      $ 3392 "'desbaste_inicial'"
      # 'desbaste_inicial'
      $ 3393 "bajada_broca≔p[0,0,-0.008,0,0,0]"
      global bajada_broca=p[0,0,-0.008,0,0,0]
      $ 3394 "bajada≔p[0,0,0.008,0,0,0]"
      global bajada=p[0,0,0.008,0,0,0]
      $ 3395 "Direction: Base Z-"
      global move_thread_flag_3395=0
      thread move_thread_3395():
        enter_critical
        move_thread_flag_3395 = 1
        local towardsPos=calculate_point_to_move_towards(p[0.0,0.0,0.0,0.0,0.0,0.0], [0.0,0.0,-1.0], 0.08)
        movel(towardsPos, a=0.035, v=0.03)
        move_thread_flag_3395 = 2
        exit_critical
      end
      move_thread_flag_3395 = 0
      move_thread_han_3395 = run move_thread_3395()
      while (True):
        sleep(1.0E-10)
        if (move_thread_flag_3395 > 1):
          join move_thread_han_3395
          $ 3396 "Until (distance)"
          break
        end
        sync()
      end
      $ 3397 "Popup: punto contacto alanzdo"
      popup("punto contacto alanzdo", "Mensaje", False, False, blocking=True)
      $ 3398 "Direction: Base Z+"
      global move_thread_flag_3398=0
      thread move_thread_3398():
        enter_critical
        move_thread_flag_3398 = 1
        local towardsPos=calculate_point_to_move_towards(p[0.0,0.0,0.0,0.0,0.0,0.0], [0.0,0.0,1.0], 0.002)
        movel(towardsPos, a=0.005, v=0.003)
        move_thread_flag_3398 = 2
        exit_critical
      end
      move_thread_flag_3398 = 0
      move_thread_han_3398 = run move_thread_3398()
      while (True):
        sleep(1.0E-10)
        if (move_thread_flag_3398 > 1):
          join move_thread_han_3398
          $ 3399 "Until (distance)"
          break
        end
        sync()
      end
      $ 3400 "Wait: 0.3"
      sleep(0.3)
      $ 3401 "Set CO[1]=Encender"
      set_configurable_digital_out(1, True)
      $ 3402 "Wait: 0.3"
      sleep(0.3)
      $ 3403 "Loop 3 times"
      Loop_58 = 0
      while (Loop_58 < 3):
        $ 3404 "bajar≔pose_add(get_actual_tcp_pose(), bajada_broca)"
        global bajar= pose_add ( get_actual_tcp_pose (), bajada_broca)
        $ 3405 "bajar" "breakAfter"
        movel(bajar, a=0.005, v=0.001)
        $ 3406 "subir≔pose_sub(get_actual_tcp_pose(), bajada_broca)"
        global subir= pose_sub ( get_actual_tcp_pose (), bajada_broca)
        $ 3407 "subir" "breakAfter"
        movel(subir, a=0.01, v=0.01)
        $ 3408 "bajada_broca≔pose_sub(bajada_broca, bajada)"
        global bajada_broca= pose_sub (bajada_broca, bajada)
        Loop_58 = Loop_58 + 1
      end
      $ 3409 "Direction: Base Z+"
      global move_thread_flag_3409=0
      thread move_thread_3409():
        enter_critical
        move_thread_flag_3409 = 1
        local towardsPos=calculate_point_to_move_towards(p[0.0,0.0,0.0,0.0,0.0,0.0], [0.0,0.0,1.0], 0.06)
        movel(towardsPos, a=0.035, v=0.03)
        move_thread_flag_3409 = 2
        exit_critical
      end
      move_thread_flag_3409 = 0
      move_thread_han_3409 = run move_thread_3409()
      while (True):
        sleep(1.0E-10)
        if (move_thread_flag_3409 > 1):
          join move_thread_han_3409
          $ 3410 "Until (distance)"
          break
        end
        sync()
      end
      $ 3411 "Set CO[1]=Apagar"
      set_configurable_digital_out(1, False)
      $ 3412 "barreno_actual≔barreno_actual+1"
      global barreno_actual=barreno_actual+1
      $ 3413 "If barreno_actual>barrenos_menos1"
      if (barreno_actual>barrenos_menos1):
        $ 3414 "cambiar_broca≔ True "
        global cambiar_broca=  True
      end
      $ 3415 "Call Quitar_broca"
      Quitar_broca()
      $ 3416 "Call Poner_broca"
      Poner_broca()
    end
    $ 3417 "Popup: Linea4 con chica Terminada!"
    popup("Linea4 con chica Terminada!", "Mensaje", False, False, blocking=True)
    $ 3418 "Broca_2"
    $ 3419 "Linea3"
    $ 3420 "Marcar_puntos"
    $ 3421 "MoveL"
    $ 3422 "Home3" "breakAfter"
    movel(Home3_p, a=0.5, v=0.1)
    $ 3423 "Linea3_A" "breakAfter"
    movel(Linea3_A_p, a=0.5, v=0.1)
    $ 3424 "Linea3_B" "breakAfter"
    movel(Linea3_B_p, a=0.5, v=0.1)
    $ 3425 "Linea3_C" "breakAfter"
    movel(Linea3_C_p, a=0.5, v=0.1)
    $ 3426 "Linea3_D" "breakAfter"
    movel(Linea3_D_p, a=0.5, v=0.1)
    $ 3427 "Linea3_E" "breakAfter"
    movel(Linea3_E_p, a=0.5, v=0.1)
    $ 3428 "Linea3_F" "breakAfter"
    movel(Linea3_F_p, a=0.5, v=0.1)
    $ 3429 "AB"
    $ 3430 "'desbaste_inicial'"
    # 'desbaste_inicial'
    $ 3431 "bajada_broca≔p[0,0,-0.012,0,0,0]"
    global bajada_broca=p[0,0,-0.012,0,0,0]
    $ 3432 "barrenos_menos1≔8"
    global barrenos_menos1=8
    $ 3433 "barreno_actual≔0"
    global barreno_actual=0
    $ 3434 "Loop barreno_actual≤barrenos_menos1"
    while (barreno_actual <= barrenos_menos1):
      $ 3435 "Perforacion"
      $ 3436 "MoveL"
      $ 3437 "internos≔interpolate_pose(Linea3_A, Linea3_B, barreno_actual/barrenos_menos1)"
      global internos= interpolate_pose (Linea3_A_p, Linea3_B_p, barreno_actual/barrenos_menos1)
      $ 3438 "internos" "breakAfter"
      movel(internos, a=0.5, v=0.1)
      $ 3439 "'desbaste_inicial'"
      # 'desbaste_inicial'
      $ 3440 "bajada_broca≔p[0,0,-0.012,0,0,0]"
      global bajada_broca=p[0,0,-0.012,0,0,0]
      $ 3441 "bajada≔p[0,0,0.012,0,0,0]"
      global bajada=p[0,0,0.012,0,0,0]
      $ 3442 "Direction: Base Z-"
      global move_thread_flag_3442=0
      thread move_thread_3442():
        enter_critical
        move_thread_flag_3442 = 1
        local towardsPos=calculate_point_to_move_towards(p[0.0,0.0,0.0,0.0,0.0,0.0], [0.0,0.0,-1.0], 0.08)
        movel(towardsPos, a=0.035, v=0.03)
        move_thread_flag_3442 = 2
        exit_critical
      end
      move_thread_flag_3442 = 0
      move_thread_han_3442 = run move_thread_3442()
      while (True):
        sleep(1.0E-10)
        if (move_thread_flag_3442 > 1):
          join move_thread_han_3442
          $ 3443 "Until (distance)"
          break
        end
        sync()
      end
      $ 3444 "Popup: punto contacto alanzdo"
      popup("punto contacto alanzdo", "Mensaje", False, False, blocking=True)
      $ 3445 "Direction: Base Z+"
      global move_thread_flag_3445=0
      thread move_thread_3445():
        enter_critical
        move_thread_flag_3445 = 1
        local towardsPos=calculate_point_to_move_towards(p[0.0,0.0,0.0,0.0,0.0,0.0], [0.0,0.0,1.0], 0.002)
        movel(towardsPos, a=0.005, v=0.003)
        move_thread_flag_3445 = 2
        exit_critical
      end
      move_thread_flag_3445 = 0
      move_thread_han_3445 = run move_thread_3445()
      while (True):
        sleep(1.0E-10)
        if (move_thread_flag_3445 > 1):
          join move_thread_han_3445
          $ 3446 "Until (distance)"
          break
        end
        sync()
      end
      $ 3447 "Wait: 0.3"
      sleep(0.3)
      $ 3448 "Set CO[1]=Encender"
      set_configurable_digital_out(1, True)
      $ 3449 "Wait: 0.3"
      sleep(0.3)
      $ 3450 "Loop 2 times"
      Loop_60 = 0
      while (Loop_60 < 2):
        $ 3451 "bajar≔pose_add(get_actual_tcp_pose(), bajada_broca)"
        global bajar= pose_add ( get_actual_tcp_pose (), bajada_broca)
        $ 3452 "bajar" "breakAfter"
        movel(bajar, a=0.005, v=0.001)
        $ 3453 "subir≔pose_sub(get_actual_tcp_pose(), bajada_broca)"
        global subir= pose_sub ( get_actual_tcp_pose (), bajada_broca)
        $ 3454 "subir" "breakAfter"
        movel(subir, a=0.01, v=0.01)
        $ 3455 "bajada_broca≔pose_sub(bajada_broca, bajada)"
        global bajada_broca= pose_sub (bajada_broca, bajada)
        Loop_60 = Loop_60 + 1
      end
      $ 3456 "Direction: Base Z+"
      global move_thread_flag_3456=0
      thread move_thread_3456():
        enter_critical
        move_thread_flag_3456 = 1
        local towardsPos=calculate_point_to_move_towards(p[0.0,0.0,0.0,0.0,0.0,0.0], [0.0,0.0,1.0], 0.06)
        movel(towardsPos, a=0.035, v=0.03)
        move_thread_flag_3456 = 2
        exit_critical
      end
      move_thread_flag_3456 = 0
      move_thread_han_3456 = run move_thread_3456()
      while (True):
        sleep(1.0E-10)
        if (move_thread_flag_3456 > 1):
          join move_thread_han_3456
          $ 3457 "Until (distance)"
          break
        end
        sync()
      end
      $ 3458 "Set CO[1]=Apagar"
      set_configurable_digital_out(1, False)
      $ 3459 "barreno_actual≔barreno_actual+1"
      global barreno_actual=barreno_actual+1
      $ 3460 "Call Quitar_broca"
      Quitar_broca()
      $ 3461 "Call Poner_broca"
      Poner_broca()
    end
    $ 3462 "CD"
    $ 3463 "'desbaste_inicial'"
    # 'desbaste_inicial'
    $ 3464 "bajada_broca≔p[0,0,-0.012,0,0,0]"
    global bajada_broca=p[0,0,-0.012,0,0,0]
    $ 3465 "barrenos_menos1≔8"
    global barrenos_menos1=8
    $ 3466 "barreno_actual≔0"
    global barreno_actual=0
    $ 3467 "Loop barreno_actual≤barrenos_menos1"
    while (barreno_actual <= barrenos_menos1):
      $ 3468 "Perforacion"
      $ 3469 "MoveL"
      $ 3470 "internos≔interpolate_pose(Linea3_C, Linea3_D, barreno_actual/barrenos_menos1)"
      global internos= interpolate_pose (Linea3_C_p, Linea3_D_p, barreno_actual/barrenos_menos1)
      $ 3471 "internos" "breakAfter"
      movel(internos, a=0.5, v=0.1)
      $ 3472 "'desbaste_inicial'"
      # 'desbaste_inicial'
      $ 3473 "bajada_broca≔p[0,0,-0.012,0,0,0]"
      global bajada_broca=p[0,0,-0.012,0,0,0]
      $ 3474 "bajada≔p[0,0,0.012,0,0,0]"
      global bajada=p[0,0,0.012,0,0,0]
      $ 3475 "Direction: Base Z-"
      global move_thread_flag_3475=0
      thread move_thread_3475():
        enter_critical
        move_thread_flag_3475 = 1
        local towardsPos=calculate_point_to_move_towards(p[0.0,0.0,0.0,0.0,0.0,0.0], [0.0,0.0,-1.0], 0.08)
        movel(towardsPos, a=0.035, v=0.03)
        move_thread_flag_3475 = 2
        exit_critical
      end
      move_thread_flag_3475 = 0
      move_thread_han_3475 = run move_thread_3475()
      while (True):
        sleep(1.0E-10)
        if (move_thread_flag_3475 > 1):
          join move_thread_han_3475
          $ 3476 "Until (distance)"
          break
        end
        sync()
      end
      $ 3477 "Popup: punto contacto alanzdo"
      popup("punto contacto alanzdo", "Mensaje", False, False, blocking=True)
      $ 3478 "Direction: Base Z+"
      global move_thread_flag_3478=0
      thread move_thread_3478():
        enter_critical
        move_thread_flag_3478 = 1
        local towardsPos=calculate_point_to_move_towards(p[0.0,0.0,0.0,0.0,0.0,0.0], [0.0,0.0,1.0], 0.002)
        movel(towardsPos, a=0.005, v=0.003)
        move_thread_flag_3478 = 2
        exit_critical
      end
      move_thread_flag_3478 = 0
      move_thread_han_3478 = run move_thread_3478()
      while (True):
        sleep(1.0E-10)
        if (move_thread_flag_3478 > 1):
          join move_thread_han_3478
          $ 3479 "Until (distance)"
          break
        end
        sync()
      end
      $ 3480 "Wait: 0.3"
      sleep(0.3)
      $ 3481 "Set CO[1]=Encender"
      set_configurable_digital_out(1, True)
      $ 3482 "Wait: 0.3"
      sleep(0.3)
      $ 3483 "Loop 2 times"
      Loop_64 = 0
      while (Loop_64 < 2):
        $ 3484 "bajar≔pose_add(get_actual_tcp_pose(), bajada_broca)"
        global bajar= pose_add ( get_actual_tcp_pose (), bajada_broca)
        $ 3485 "bajar" "breakAfter"
        movel(bajar, a=0.005, v=0.001)
        $ 3486 "subir≔pose_sub(get_actual_tcp_pose(), bajada_broca)"
        global subir= pose_sub ( get_actual_tcp_pose (), bajada_broca)
        $ 3487 "subir" "breakAfter"
        movel(subir, a=0.01, v=0.01)
        $ 3488 "bajada_broca≔pose_sub(bajada_broca, bajada)"
        global bajada_broca= pose_sub (bajada_broca, bajada)
        Loop_64 = Loop_64 + 1
      end
      $ 3489 "Direction: Base Z+"
      global move_thread_flag_3489=0
      thread move_thread_3489():
        enter_critical
        move_thread_flag_3489 = 1
        local towardsPos=calculate_point_to_move_towards(p[0.0,0.0,0.0,0.0,0.0,0.0], [0.0,0.0,1.0], 0.06)
        movel(towardsPos, a=0.035, v=0.03)
        move_thread_flag_3489 = 2
        exit_critical
      end
      move_thread_flag_3489 = 0
      move_thread_han_3489 = run move_thread_3489()
      while (True):
        sleep(1.0E-10)
        if (move_thread_flag_3489 > 1):
          join move_thread_han_3489
          $ 3490 "Until (distance)"
          break
        end
        sync()
      end
      $ 3491 "Set CO[1]=Apagar"
      set_configurable_digital_out(1, False)
      $ 3492 "barreno_actual≔barreno_actual+1"
      global barreno_actual=barreno_actual+1
      $ 3493 "Call Quitar_broca"
      Quitar_broca()
      $ 3494 "Call Poner_broca"
      Poner_broca()
    end
    $ 3495 "EF"
    $ 3496 "'desbaste_inicial'"
    # 'desbaste_inicial'
    $ 3497 "bajada_broca≔p[0,0,-0.012,0,0,0]"
    global bajada_broca=p[0,0,-0.012,0,0,0]
    $ 3498 "barrenos_menos1≔8"
    global barrenos_menos1=8
    $ 3499 "barreno_actual≔0"
    global barreno_actual=0
    $ 3500 "Loop barreno_actual≤barrenos_menos1"
    while (barreno_actual <= barrenos_menos1):
      $ 3501 "Perforacion"
      $ 3502 "MoveL"
      $ 3503 "internos≔interpolate_pose(Linea3_E, Linea3_F, barreno_actual/barrenos_menos1)"
      global internos= interpolate_pose (Linea3_E_p, Linea3_F_p, barreno_actual/barrenos_menos1)
      $ 3504 "internos" "breakAfter"
      movel(internos, a=0.5, v=0.1)
      $ 3505 "'desbaste_inicial'"
      # 'desbaste_inicial'
      $ 3506 "bajada_broca≔p[0,0,-0.012,0,0,0]"
      global bajada_broca=p[0,0,-0.012,0,0,0]
      $ 3507 "bajada≔p[0,0,0.012,0,0,0]"
      global bajada=p[0,0,0.012,0,0,0]
      $ 3508 "Direction: Base Z-"
      global move_thread_flag_3508=0
      thread move_thread_3508():
        enter_critical
        move_thread_flag_3508 = 1
        local towardsPos=calculate_point_to_move_towards(p[0.0,0.0,0.0,0.0,0.0,0.0], [0.0,0.0,-1.0], 0.08)
        movel(towardsPos, a=0.035, v=0.03)
        move_thread_flag_3508 = 2
        exit_critical
      end
      move_thread_flag_3508 = 0
      move_thread_han_3508 = run move_thread_3508()
      while (True):
        sleep(1.0E-10)
        if (move_thread_flag_3508 > 1):
          join move_thread_han_3508
          $ 3509 "Until (distance)"
          break
        end
        sync()
      end
      $ 3510 "Popup: punto contacto alanzdo"
      popup("punto contacto alanzdo", "Mensaje", False, False, blocking=True)
      $ 3511 "Direction: Base Z+"
      global move_thread_flag_3511=0
      thread move_thread_3511():
        enter_critical
        move_thread_flag_3511 = 1
        local towardsPos=calculate_point_to_move_towards(p[0.0,0.0,0.0,0.0,0.0,0.0], [0.0,0.0,1.0], 0.002)
        movel(towardsPos, a=0.005, v=0.003)
        move_thread_flag_3511 = 2
        exit_critical
      end
      move_thread_flag_3511 = 0
      move_thread_han_3511 = run move_thread_3511()
      while (True):
        sleep(1.0E-10)
        if (move_thread_flag_3511 > 1):
          join move_thread_han_3511
          $ 3512 "Until (distance)"
          break
        end
        sync()
      end
      $ 3513 "Wait: 0.3"
      sleep(0.3)
      $ 3514 "Set CO[1]=Encender"
      set_configurable_digital_out(1, True)
      $ 3515 "Wait: 0.3"
      sleep(0.3)
      $ 3516 "Loop 2 times"
      Loop_68 = 0
      while (Loop_68 < 2):
        $ 3517 "bajar≔pose_add(get_actual_tcp_pose(), bajada_broca)"
        global bajar= pose_add ( get_actual_tcp_pose (), bajada_broca)
        $ 3518 "bajar" "breakAfter"
        movel(bajar, a=0.005, v=0.001)
        $ 3519 "subir≔pose_sub(get_actual_tcp_pose(), bajada_broca)"
        global subir= pose_sub ( get_actual_tcp_pose (), bajada_broca)
        $ 3520 "subir" "breakAfter"
        movel(subir, a=0.01, v=0.01)
        $ 3521 "bajada_broca≔pose_sub(bajada_broca, bajada)"
        global bajada_broca= pose_sub (bajada_broca, bajada)
        Loop_68 = Loop_68 + 1
      end
      $ 3522 "Direction: Base Z+"
      global move_thread_flag_3522=0
      thread move_thread_3522():
        enter_critical
        move_thread_flag_3522 = 1
        local towardsPos=calculate_point_to_move_towards(p[0.0,0.0,0.0,0.0,0.0,0.0], [0.0,0.0,1.0], 0.06)
        movel(towardsPos, a=0.035, v=0.03)
        move_thread_flag_3522 = 2
        exit_critical
      end
      move_thread_flag_3522 = 0
      move_thread_han_3522 = run move_thread_3522()
      while (True):
        sleep(1.0E-10)
        if (move_thread_flag_3522 > 1):
          join move_thread_han_3522
          $ 3523 "Until (distance)"
          break
        end
        sync()
      end
      $ 3524 "Set CO[1]=Apagar"
      set_configurable_digital_out(1, False)
      $ 3525 "barreno_actual≔barreno_actual+1"
      global barreno_actual=barreno_actual+1
      $ 3526 "Call Quitar_broca"
      Quitar_broca()
      $ 3527 "Call Poner_broca"
      Poner_broca()
    end
    $ 3528 "Popup: Linea3 con media Terminada!"
    popup("Linea3 con media Terminada!", "Mensaje", False, False, blocking=True)
    $ 3529 "Linea4"
    $ 3530 "Marcar_puntos"
    $ 3531 "MoveL"
    $ 3532 "Home3" "breakAfter"
    movel(Home3_p, a=0.5, v=0.1)
    $ 3533 "Linea4_A" "breakAfter"
    movel(Linea4_A_p, a=0.5, v=0.1)
    $ 3534 "Linea4_B" "breakAfter"
    movel(Linea4_B_p, a=0.5, v=0.1)
    $ 3535 "Linea4_C" "breakAfter"
    movel(Linea4_C_p, a=0.5, v=0.1)
    $ 3536 "Linea4_D" "breakAfter"
    movel(Linea4_D_p, a=0.5, v=0.1)
    $ 3537 "Linea4_E" "breakAfter"
    movel(Linea4_E_p, a=0.5, v=0.1)
    $ 3538 "Linea4_F" "breakAfter"
    movel(Linea4_F_p, a=0.5, v=0.1)
    $ 3539 "AB"
    $ 3540 "'desbaste_inicial'"
    # 'desbaste_inicial'
    $ 3541 "bajada_broca≔p[0,0,-0.012,0,0,0]"
    global bajada_broca=p[0,0,-0.012,0,0,0]
    $ 3542 "barrenos_menos1≔8"
    global barrenos_menos1=8
    $ 3543 "barreno_actual≔0"
    global barreno_actual=0
    $ 3544 "Loop barreno_actual≤barrenos_menos1"
    while (barreno_actual <= barrenos_menos1):
      $ 3545 "Perforacion"
      $ 3546 "MoveL"
      $ 3547 "internos≔interpolate_pose(Linea4_A, Linea4_B, barreno_actual/barrenos_menos1)"
      global internos= interpolate_pose (Linea4_A_p, Linea4_B_p, barreno_actual/barrenos_menos1)
      $ 3548 "internos" "breakAfter"
      movel(internos, a=0.5, v=0.1)
      $ 3549 "'desbaste_inicial'"
      # 'desbaste_inicial'
      $ 3550 "bajada_broca≔p[0,0,-0.012,0,0,0]"
      global bajada_broca=p[0,0,-0.012,0,0,0]
      $ 3551 "bajada≔p[0,0,0.012,0,0,0]"
      global bajada=p[0,0,0.012,0,0,0]
      $ 3552 "Direction: Base Z-"
      global move_thread_flag_3552=0
      thread move_thread_3552():
        enter_critical
        move_thread_flag_3552 = 1
        local towardsPos=calculate_point_to_move_towards(p[0.0,0.0,0.0,0.0,0.0,0.0], [0.0,0.0,-1.0], 0.08)
        movel(towardsPos, a=0.035, v=0.03)
        move_thread_flag_3552 = 2
        exit_critical
      end
      move_thread_flag_3552 = 0
      move_thread_han_3552 = run move_thread_3552()
      while (True):
        sleep(1.0E-10)
        if (move_thread_flag_3552 > 1):
          join move_thread_han_3552
          $ 3553 "Until (distance)"
          break
        end
        sync()
      end
      $ 3554 "Popup: punto contacto alanzdo"
      popup("punto contacto alanzdo", "Mensaje", False, False, blocking=True)
      $ 3555 "Direction: Base Z+"
      global move_thread_flag_3555=0
      thread move_thread_3555():
        enter_critical
        move_thread_flag_3555 = 1
        local towardsPos=calculate_point_to_move_towards(p[0.0,0.0,0.0,0.0,0.0,0.0], [0.0,0.0,1.0], 0.002)
        movel(towardsPos, a=0.005, v=0.003)
        move_thread_flag_3555 = 2
        exit_critical
      end
      move_thread_flag_3555 = 0
      move_thread_han_3555 = run move_thread_3555()
      while (True):
        sleep(1.0E-10)
        if (move_thread_flag_3555 > 1):
          join move_thread_han_3555
          $ 3556 "Until (distance)"
          break
        end
        sync()
      end
      $ 3557 "Wait: 0.3"
      sleep(0.3)
      $ 3558 "Set CO[1]=Encender"
      set_configurable_digital_out(1, True)
      $ 3559 "Wait: 0.3"
      sleep(0.3)
      $ 3560 "Loop 2 times"
      Loop_72 = 0
      while (Loop_72 < 2):
        $ 3561 "bajar≔pose_add(get_actual_tcp_pose(), bajada_broca)"
        global bajar= pose_add ( get_actual_tcp_pose (), bajada_broca)
        $ 3562 "bajar" "breakAfter"
        movel(bajar, a=0.005, v=0.001)
        $ 3563 "subir≔pose_sub(get_actual_tcp_pose(), bajada_broca)"
        global subir= pose_sub ( get_actual_tcp_pose (), bajada_broca)
        $ 3564 "subir" "breakAfter"
        movel(subir, a=0.01, v=0.01)
        $ 3565 "bajada_broca≔pose_sub(bajada_broca, bajada)"
        global bajada_broca= pose_sub (bajada_broca, bajada)
        Loop_72 = Loop_72 + 1
      end
      $ 3566 "Direction: Base Z+"
      global move_thread_flag_3566=0
      thread move_thread_3566():
        enter_critical
        move_thread_flag_3566 = 1
        local towardsPos=calculate_point_to_move_towards(p[0.0,0.0,0.0,0.0,0.0,0.0], [0.0,0.0,1.0], 0.06)
        movel(towardsPos, a=0.035, v=0.03)
        move_thread_flag_3566 = 2
        exit_critical
      end
      move_thread_flag_3566 = 0
      move_thread_han_3566 = run move_thread_3566()
      while (True):
        sleep(1.0E-10)
        if (move_thread_flag_3566 > 1):
          join move_thread_han_3566
          $ 3567 "Until (distance)"
          break
        end
        sync()
      end
      $ 3568 "Set CO[1]=Apagar"
      set_configurable_digital_out(1, False)
      $ 3569 "barreno_actual≔barreno_actual+1"
      global barreno_actual=barreno_actual+1
      $ 3570 "Call Quitar_broca"
      Quitar_broca()
      $ 3571 "Call Poner_broca"
      Poner_broca()
    end
    $ 3572 "CD"
    $ 3573 "'desbaste_inicial'"
    # 'desbaste_inicial'
    $ 3574 "bajada_broca≔p[0,0,-0.012,0,0,0]"
    global bajada_broca=p[0,0,-0.012,0,0,0]
    $ 3575 "barrenos_menos1≔8"
    global barrenos_menos1=8
    $ 3576 "barreno_actual≔0"
    global barreno_actual=0
    $ 3577 "Loop barreno_actual≤barrenos_menos1"
    while (barreno_actual <= barrenos_menos1):
      $ 3578 "Perforacion"
      $ 3579 "MoveL"
      $ 3580 "internos≔interpolate_pose(Linea4_C, Linea4_D, barreno_actual/barrenos_menos1)"
      global internos= interpolate_pose (Linea4_C_p, Linea4_D_p, barreno_actual/barrenos_menos1)
      $ 3581 "internos" "breakAfter"
      movel(internos, a=0.5, v=0.1)
      $ 3582 "'desbaste_inicial'"
      # 'desbaste_inicial'
      $ 3583 "bajada_broca≔p[0,0,-0.012,0,0,0]"
      global bajada_broca=p[0,0,-0.012,0,0,0]
      $ 3584 "bajada≔p[0,0,0.012,0,0,0]"
      global bajada=p[0,0,0.012,0,0,0]
      $ 3585 "Direction: Base Z-"
      global move_thread_flag_3585=0
      thread move_thread_3585():
        enter_critical
        move_thread_flag_3585 = 1
        local towardsPos=calculate_point_to_move_towards(p[0.0,0.0,0.0,0.0,0.0,0.0], [0.0,0.0,-1.0], 0.08)
        movel(towardsPos, a=0.035, v=0.03)
        move_thread_flag_3585 = 2
        exit_critical
      end
      move_thread_flag_3585 = 0
      move_thread_han_3585 = run move_thread_3585()
      while (True):
        sleep(1.0E-10)
        if (move_thread_flag_3585 > 1):
          join move_thread_han_3585
          $ 3586 "Until (distance)"
          break
        end
        sync()
      end
      $ 3587 "Popup: punto contacto alanzdo"
      popup("punto contacto alanzdo", "Mensaje", False, False, blocking=True)
      $ 3588 "Direction: Base Z+"
      global move_thread_flag_3588=0
      thread move_thread_3588():
        enter_critical
        move_thread_flag_3588 = 1
        local towardsPos=calculate_point_to_move_towards(p[0.0,0.0,0.0,0.0,0.0,0.0], [0.0,0.0,1.0], 0.002)
        movel(towardsPos, a=0.005, v=0.003)
        move_thread_flag_3588 = 2
        exit_critical
      end
      move_thread_flag_3588 = 0
      move_thread_han_3588 = run move_thread_3588()
      while (True):
        sleep(1.0E-10)
        if (move_thread_flag_3588 > 1):
          join move_thread_han_3588
          $ 3589 "Until (distance)"
          break
        end
        sync()
      end
      $ 3590 "Wait: 0.3"
      sleep(0.3)
      $ 3591 "Set CO[1]=Encender"
      set_configurable_digital_out(1, True)
      $ 3592 "Wait: 0.3"
      sleep(0.3)
      $ 3593 "Loop 2 times"
      Loop_77 = 0
      while (Loop_77 < 2):
        $ 3594 "bajar≔pose_add(get_actual_tcp_pose(), bajada_broca)"
        global bajar= pose_add ( get_actual_tcp_pose (), bajada_broca)
        $ 3595 "bajar" "breakAfter"
        movel(bajar, a=0.005, v=0.001)
        $ 3596 "subir≔pose_sub(get_actual_tcp_pose(), bajada_broca)"
        global subir= pose_sub ( get_actual_tcp_pose (), bajada_broca)
        $ 3597 "subir" "breakAfter"
        movel(subir, a=0.01, v=0.01)
        $ 3598 "bajada_broca≔pose_sub(bajada_broca, bajada)"
        global bajada_broca= pose_sub (bajada_broca, bajada)
        Loop_77 = Loop_77 + 1
      end
      $ 3599 "Direction: Base Z+"
      global move_thread_flag_3599=0
      thread move_thread_3599():
        enter_critical
        move_thread_flag_3599 = 1
        local towardsPos=calculate_point_to_move_towards(p[0.0,0.0,0.0,0.0,0.0,0.0], [0.0,0.0,1.0], 0.06)
        movel(towardsPos, a=0.035, v=0.03)
        move_thread_flag_3599 = 2
        exit_critical
      end
      move_thread_flag_3599 = 0
      move_thread_han_3599 = run move_thread_3599()
      while (True):
        sleep(1.0E-10)
        if (move_thread_flag_3599 > 1):
          join move_thread_han_3599
          $ 3600 "Until (distance)"
          break
        end
        sync()
      end
      $ 3601 "Set CO[1]=Apagar"
      set_configurable_digital_out(1, False)
      $ 3602 "barreno_actual≔barreno_actual+1"
      global barreno_actual=barreno_actual+1
      $ 3603 "Call Quitar_broca"
      Quitar_broca()
      $ 3604 "Call Poner_broca"
      Poner_broca()
    end
    $ 3605 "EF"
    $ 3606 "'desbaste_inicial'"
    # 'desbaste_inicial'
    $ 3607 "bajada_broca≔p[0,0,-0.012,0,0,0]"
    global bajada_broca=p[0,0,-0.012,0,0,0]
    $ 3608 "barrenos_menos1≔8"
    global barrenos_menos1=8
    $ 3609 "barreno_actual≔0"
    global barreno_actual=0
    $ 3610 "Loop barreno_actual≤barrenos_menos1"
    while (barreno_actual <= barrenos_menos1):
      $ 3611 "Perforacion"
      $ 3612 "MoveL"
      $ 3613 "internos≔interpolate_pose(Linea4_E, Linea4_F, barreno_actual/barrenos_menos1)"
      global internos= interpolate_pose (Linea4_E_p, Linea4_F_p, barreno_actual/barrenos_menos1)
      $ 3614 "internos" "breakAfter"
      movel(internos, a=0.5, v=0.1)
      $ 3615 "'desbaste_inicial'"
      # 'desbaste_inicial'
      $ 3616 "bajada_broca≔p[0,0,-0.012,0,0,0]"
      global bajada_broca=p[0,0,-0.012,0,0,0]
      $ 3617 "bajada≔p[0,0,0.012,0,0,0]"
      global bajada=p[0,0,0.012,0,0,0]
      $ 3618 "Direction: Base Z-"
      global move_thread_flag_3618=0
      thread move_thread_3618():
        enter_critical
        move_thread_flag_3618 = 1
        local towardsPos=calculate_point_to_move_towards(p[0.0,0.0,0.0,0.0,0.0,0.0], [0.0,0.0,-1.0], 0.08)
        movel(towardsPos, a=0.035, v=0.03)
        move_thread_flag_3618 = 2
        exit_critical
      end
      move_thread_flag_3618 = 0
      move_thread_han_3618 = run move_thread_3618()
      while (True):
        sleep(1.0E-10)
        if (move_thread_flag_3618 > 1):
          join move_thread_han_3618
          $ 3619 "Until (distance)"
          break
        end
        sync()
      end
      $ 3620 "Popup: punto contacto alanzdo"
      popup("punto contacto alanzdo", "Mensaje", False, False, blocking=True)
      $ 3621 "Direction: Base Z+"
      global move_thread_flag_3621=0
      thread move_thread_3621():
        enter_critical
        move_thread_flag_3621 = 1
        local towardsPos=calculate_point_to_move_towards(p[0.0,0.0,0.0,0.0,0.0,0.0], [0.0,0.0,1.0], 0.002)
        movel(towardsPos, a=0.005, v=0.003)
        move_thread_flag_3621 = 2
        exit_critical
      end
      move_thread_flag_3621 = 0
      move_thread_han_3621 = run move_thread_3621()
      while (True):
        sleep(1.0E-10)
        if (move_thread_flag_3621 > 1):
          join move_thread_han_3621
          $ 3622 "Until (distance)"
          break
        end
        sync()
      end
      $ 3623 "Wait: 0.3"
      sleep(0.3)
      $ 3624 "Set CO[1]=Encender"
      set_configurable_digital_out(1, True)
      $ 3625 "Wait: 0.3"
      sleep(0.3)
      $ 3626 "Loop 2 times"
      Loop_81 = 0
      while (Loop_81 < 2):
        $ 3627 "bajar≔pose_add(get_actual_tcp_pose(), bajada_broca)"
        global bajar= pose_add ( get_actual_tcp_pose (), bajada_broca)
        $ 3628 "bajar" "breakAfter"
        movel(bajar, a=0.005, v=0.001)
        $ 3629 "subir≔pose_sub(get_actual_tcp_pose(), bajada_broca)"
        global subir= pose_sub ( get_actual_tcp_pose (), bajada_broca)
        $ 3630 "subir" "breakAfter"
        movel(subir, a=0.01, v=0.01)
        $ 3631 "bajada_broca≔pose_sub(bajada_broca, bajada)"
        global bajada_broca= pose_sub (bajada_broca, bajada)
        Loop_81 = Loop_81 + 1
      end
      $ 3632 "Direction: Base Z+"
      global move_thread_flag_3632=0
      thread move_thread_3632():
        enter_critical
        move_thread_flag_3632 = 1
        local towardsPos=calculate_point_to_move_towards(p[0.0,0.0,0.0,0.0,0.0,0.0], [0.0,0.0,1.0], 0.06)
        movel(towardsPos, a=0.035, v=0.03)
        move_thread_flag_3632 = 2
        exit_critical
      end
      move_thread_flag_3632 = 0
      move_thread_han_3632 = run move_thread_3632()
      while (True):
        sleep(1.0E-10)
        if (move_thread_flag_3632 > 1):
          join move_thread_han_3632
          $ 3633 "Until (distance)"
          break
        end
        sync()
      end
      $ 3634 "Set CO[1]=Apagar"
      set_configurable_digital_out(1, False)
      $ 3635 "barreno_actual≔barreno_actual+1"
      global barreno_actual=barreno_actual+1
      $ 3636 "If barreno_actual>barrenos_menos1"
      if (barreno_actual>barrenos_menos1):
        $ 3637 "cambiar_broca≔ True "
        global cambiar_broca=  True
      end
      $ 3638 "Call Quitar_broca"
      Quitar_broca()
      $ 3639 "Call Poner_broca"
      Poner_broca()
    end
    $ 3640 "Popup: Linea4 con media Terminada!"
    popup("Linea4 con media Terminada!", "Mensaje", False, False, blocking=True)
    $ 3641 "Broca_3"
    $ 3642 "Linea3"
    $ 3643 "Marcar_puntos"
    $ 3644 "MoveL"
    $ 3645 "Home3" "breakAfter"
    movel(Home3_p, a=0.5, v=0.1)
    $ 3646 "var"
    $ 3647 "barrenos_hechos≔0"
    global barrenos_hechos=0
    $ 3648 "eje7≔3"
    global eje7=3
    $ 3649 "cambiar_broca≔ False "
    global cambiar_broca=  False
    $ 3650 "iniciando_prog≔ True "
    global iniciando_prog=  True
    $ 3651 "Call Poner_broca"
    Poner_broca()
    $ 3652 "Linea3_A" "breakAfter"
    movel(Linea3_A_p, a=0.5, v=0.1)
    $ 3653 "Linea3_B" "breakAfter"
    movel(Linea3_B_p, a=0.5, v=0.1)
    $ 3654 "Linea3_C" "breakAfter"
    movel(Linea3_C_p, a=0.5, v=0.1)
    $ 3655 "Linea3_D" "breakAfter"
    movel(Linea3_D_p, a=0.5, v=0.1)
    $ 3656 "Linea3_E" "breakAfter"
    movel(Linea3_E_p, a=0.5, v=0.1)
    $ 3657 "Linea3_F" "breakAfter"
    movel(Linea3_F_p, a=0.5, v=0.1)
    $ 3658 "AB"
    $ 3659 "'desbaste_inicial'"
    # 'desbaste_inicial'
    $ 3660 "bajada_broca≔p[0,0,-0.024,0,0,0]"
    global bajada_broca=p[0,0,-0.024,0,0,0]
    $ 3661 "barrenos_menos1≔8"
    global barrenos_menos1=8
    $ 3662 "barreno_actual≔5"
    global barreno_actual=5
    $ 3663 "Loop barreno_actual≤barrenos_menos1"
    while (barreno_actual <= barrenos_menos1):
      $ 3664 "Perforacion"
      $ 3665 "MoveL"
      $ 3666 "internos≔interpolate_pose(Linea3_A, Linea3_B, barreno_actual/barrenos_menos1)"
      global internos= interpolate_pose (Linea3_A_p, Linea3_B_p, barreno_actual/barrenos_menos1)
      $ 3667 "internos" "breakAfter"
      movel(internos, a=0.5, v=0.1)
      $ 3668 "'desbaste_inicial'"
      # 'desbaste_inicial'
      $ 3669 "bajada_broca≔p[0,0,-0.024,0,0,0]"
      global bajada_broca=p[0,0,-0.024,0,0,0]
      $ 3670 "bajada≔p[0,0,0.024,0,0,0]"
      global bajada=p[0,0,0.024,0,0,0]
      $ 3671 "Direction: Base Z-"
      global move_thread_flag_3671=0
      thread move_thread_3671():
        enter_critical
        move_thread_flag_3671 = 1
        local towardsPos=calculate_point_to_move_towards(p[0.0,0.0,0.0,0.0,0.0,0.0], [0.0,0.0,-1.0], 0.083)
        movel(towardsPos, a=0.035, v=0.03)
        move_thread_flag_3671 = 2
        exit_critical
      end
      move_thread_flag_3671 = 0
      move_thread_han_3671 = run move_thread_3671()
      while (True):
        sleep(1.0E-10)
        if (move_thread_flag_3671 > 1):
          join move_thread_han_3671
          $ 3672 "Until (distance)"
          break
        end
        sync()
      end
      $ 3673 "Popup: punto contacto alanzdo"
      popup("punto contacto alanzdo", "Mensaje", False, False, blocking=True)
      $ 3674 "Direction: Base Z+"
      global move_thread_flag_3674=0
      thread move_thread_3674():
        enter_critical
        move_thread_flag_3674 = 1
        local towardsPos=calculate_point_to_move_towards(p[0.0,0.0,0.0,0.0,0.0,0.0], [0.0,0.0,1.0], 0.002)
        movel(towardsPos, a=0.005, v=0.003)
        move_thread_flag_3674 = 2
        exit_critical
      end
      move_thread_flag_3674 = 0
      move_thread_han_3674 = run move_thread_3674()
      while (True):
        sleep(1.0E-10)
        if (move_thread_flag_3674 > 1):
          join move_thread_han_3674
          $ 3675 "Until (distance)"
          break
        end
        sync()
      end
      $ 3676 "Wait: 0.3"
      sleep(0.3)
      $ 3677 "Set CO[1]=Encender"
      set_configurable_digital_out(1, True)
      $ 3678 "Wait: 0.3"
      sleep(0.3)
      $ 3679 "Loop 1 times"
      Loop_86 = 0
      while (Loop_86 < 1):
        $ 3680 "bajar≔pose_add(get_actual_tcp_pose(), bajada_broca)"
        global bajar= pose_add ( get_actual_tcp_pose (), bajada_broca)
        $ 3681 "bajar" "breakAfter"
        movel(bajar, a=0.005, v=0.001)
        $ 3682 "subir≔pose_sub(get_actual_tcp_pose(), bajada_broca)"
        global subir= pose_sub ( get_actual_tcp_pose (), bajada_broca)
        $ 3683 "subir" "breakAfter"
        movel(subir, a=0.01, v=0.01)
        $ 3684 "bajada_broca≔pose_sub(bajada_broca, bajada)"
        global bajada_broca= pose_sub (bajada_broca, bajada)
        Loop_86 = Loop_86 + 1
      end
      $ 3685 "Direction: Base Z+"
      global move_thread_flag_3685=0
      thread move_thread_3685():
        enter_critical
        move_thread_flag_3685 = 1
        local towardsPos=calculate_point_to_move_towards(p[0.0,0.0,0.0,0.0,0.0,0.0], [0.0,0.0,1.0], 0.06)
        movel(towardsPos, a=0.035, v=0.03)
        move_thread_flag_3685 = 2
        exit_critical
      end
      move_thread_flag_3685 = 0
      move_thread_han_3685 = run move_thread_3685()
      while (True):
        sleep(1.0E-10)
        if (move_thread_flag_3685 > 1):
          join move_thread_han_3685
          $ 3686 "Until (distance)"
          break
        end
        sync()
      end
      $ 3687 "Set CO[1]=Apagar"
      set_configurable_digital_out(1, False)
      $ 3688 "barreno_actual≔barreno_actual+1"
      global barreno_actual=barreno_actual+1
      $ 3689 "Call Quitar_broca"
      Quitar_broca()
      $ 3690 "Call Poner_broca"
      Poner_broca()
    end
    $ 3691 "CD"
    $ 3692 "'desbaste_inicial'"
    # 'desbaste_inicial'
    $ 3693 "bajada_broca≔p[0,0,-0.024,0,0,0]"
    global bajada_broca=p[0,0,-0.024,0,0,0]
    $ 3694 "barrenos_menos1≔8"
    global barrenos_menos1=8
    $ 3695 "barreno_actual≔0"
    global barreno_actual=0
    $ 3696 "Loop barreno_actual≤barrenos_menos1"
    while (barreno_actual <= barrenos_menos1):
      $ 3697 "Perforacion"
      $ 3698 "MoveL"
      $ 3699 "internos≔interpolate_pose(Linea3_C, Linea3_D, barreno_actual/barrenos_menos1)"
      global internos= interpolate_pose (Linea3_C_p, Linea3_D_p, barreno_actual/barrenos_menos1)
      $ 3700 "internos" "breakAfter"
      movel(internos, a=0.5, v=0.1)
      $ 3701 "'desbaste_inicial'"
      # 'desbaste_inicial'
      $ 3702 "bajada_broca≔p[0,0,-0.024,0,0,0]"
      global bajada_broca=p[0,0,-0.024,0,0,0]
      $ 3703 "bajada≔p[0,0,0.024,0,0,0]"
      global bajada=p[0,0,0.024,0,0,0]
      $ 3704 "Direction: Base Z-"
      global move_thread_flag_3704=0
      thread move_thread_3704():
        enter_critical
        move_thread_flag_3704 = 1
        local towardsPos=calculate_point_to_move_towards(p[0.0,0.0,0.0,0.0,0.0,0.0], [0.0,0.0,-1.0], 0.083)
        movel(towardsPos, a=0.035, v=0.03)
        move_thread_flag_3704 = 2
        exit_critical
      end
      move_thread_flag_3704 = 0
      move_thread_han_3704 = run move_thread_3704()
      while (True):
        sleep(1.0E-10)
        if (move_thread_flag_3704 > 1):
          join move_thread_han_3704
          $ 3705 "Until (distance)"
          break
        end
        sync()
      end
      $ 3706 "Popup: punto contacto alanzdo"
      popup("punto contacto alanzdo", "Mensaje", False, False, blocking=True)
      $ 3707 "Direction: Base Z+"
      global move_thread_flag_3707=0
      thread move_thread_3707():
        enter_critical
        move_thread_flag_3707 = 1
        local towardsPos=calculate_point_to_move_towards(p[0.0,0.0,0.0,0.0,0.0,0.0], [0.0,0.0,1.0], 0.002)
        movel(towardsPos, a=0.005, v=0.003)
        move_thread_flag_3707 = 2
        exit_critical
      end
      move_thread_flag_3707 = 0
      move_thread_han_3707 = run move_thread_3707()
      while (True):
        sleep(1.0E-10)
        if (move_thread_flag_3707 > 1):
          join move_thread_han_3707
          $ 3708 "Until (distance)"
          break
        end
        sync()
      end
      $ 3709 "Wait: 0.3"
      sleep(0.3)
      $ 3710 "Set CO[1]=Encender"
      set_configurable_digital_out(1, True)
      $ 3711 "Wait: 0.3"
      sleep(0.3)
      $ 3712 "Loop 1 times"
      Loop_91 = 0
      while (Loop_91 < 1):
        $ 3713 "bajar≔pose_add(get_actual_tcp_pose(), bajada_broca)"
        global bajar= pose_add ( get_actual_tcp_pose (), bajada_broca)
        $ 3714 "bajar" "breakAfter"
        movel(bajar, a=0.005, v=0.001)
        $ 3715 "subir≔pose_sub(get_actual_tcp_pose(), bajada_broca)"
        global subir= pose_sub ( get_actual_tcp_pose (), bajada_broca)
        $ 3716 "subir" "breakAfter"
        movel(subir, a=0.01, v=0.01)
        $ 3717 "bajada_broca≔pose_sub(bajada_broca, bajada)"
        global bajada_broca= pose_sub (bajada_broca, bajada)
        Loop_91 = Loop_91 + 1
      end
      $ 3718 "Direction: Base Z+"
      global move_thread_flag_3718=0
      thread move_thread_3718():
        enter_critical
        move_thread_flag_3718 = 1
        local towardsPos=calculate_point_to_move_towards(p[0.0,0.0,0.0,0.0,0.0,0.0], [0.0,0.0,1.0], 0.06)
        movel(towardsPos, a=0.035, v=0.03)
        move_thread_flag_3718 = 2
        exit_critical
      end
      move_thread_flag_3718 = 0
      move_thread_han_3718 = run move_thread_3718()
      while (True):
        sleep(1.0E-10)
        if (move_thread_flag_3718 > 1):
          join move_thread_han_3718
          $ 3719 "Until (distance)"
          break
        end
        sync()
      end
      $ 3720 "Set CO[1]=Apagar"
      set_configurable_digital_out(1, False)
      $ 3721 "barreno_actual≔barreno_actual+1"
      global barreno_actual=barreno_actual+1
      $ 3722 "Call Quitar_broca"
      Quitar_broca()
      $ 3723 "Call Poner_broca"
      Poner_broca()
    end
    $ 3724 "EF"
    $ 3725 "'desbaste_inicial'"
    # 'desbaste_inicial'
    $ 3726 "bajada_broca≔p[0,0,-0.024,0,0,0]"
    global bajada_broca=p[0,0,-0.024,0,0,0]
    $ 3727 "barrenos_menos1≔8"
    global barrenos_menos1=8
    $ 3728 "barreno_actual≔0"
    global barreno_actual=0
    $ 3729 "Loop barreno_actual≤barrenos_menos1"
    while (barreno_actual <= barrenos_menos1):
      $ 3730 "Perforacion"
      $ 3731 "MoveL"
      $ 3732 "internos≔interpolate_pose(Linea3_E, Linea3_F, barreno_actual/barrenos_menos1)"
      global internos= interpolate_pose (Linea3_E_p, Linea3_F_p, barreno_actual/barrenos_menos1)
      $ 3733 "internos" "breakAfter"
      movel(internos, a=0.5, v=0.1)
      $ 3734 "'desbaste_inicial'"
      # 'desbaste_inicial'
      $ 3735 "bajada_broca≔p[0,0,-0.024,0,0,0]"
      global bajada_broca=p[0,0,-0.024,0,0,0]
      $ 3736 "bajada≔p[0,0,0.024,0,0,0]"
      global bajada=p[0,0,0.024,0,0,0]
      $ 3737 "Direction: Base Z-"
      global move_thread_flag_3737=0
      thread move_thread_3737():
        enter_critical
        move_thread_flag_3737 = 1
        local towardsPos=calculate_point_to_move_towards(p[0.0,0.0,0.0,0.0,0.0,0.0], [0.0,0.0,-1.0], 0.083)
        movel(towardsPos, a=0.035, v=0.03)
        move_thread_flag_3737 = 2
        exit_critical
      end
      move_thread_flag_3737 = 0
      move_thread_han_3737 = run move_thread_3737()
      while (True):
        sleep(1.0E-10)
        if (move_thread_flag_3737 > 1):
          join move_thread_han_3737
          $ 3738 "Until (distance)"
          break
        end
        sync()
      end
      $ 3739 "Popup: punto contacto alanzdo"
      popup("punto contacto alanzdo", "Mensaje", False, False, blocking=True)
      $ 3740 "Direction: Base Z+"
      global move_thread_flag_3740=0
      thread move_thread_3740():
        enter_critical
        move_thread_flag_3740 = 1
        local towardsPos=calculate_point_to_move_towards(p[0.0,0.0,0.0,0.0,0.0,0.0], [0.0,0.0,1.0], 0.002)
        movel(towardsPos, a=0.005, v=0.003)
        move_thread_flag_3740 = 2
        exit_critical
      end
      move_thread_flag_3740 = 0
      move_thread_han_3740 = run move_thread_3740()
      while (True):
        sleep(1.0E-10)
        if (move_thread_flag_3740 > 1):
          join move_thread_han_3740
          $ 3741 "Until (distance)"
          break
        end
        sync()
      end
      $ 3742 "Wait: 0.3"
      sleep(0.3)
      $ 3743 "Set CO[1]=Encender"
      set_configurable_digital_out(1, True)
      $ 3744 "Wait: 0.3"
      sleep(0.3)
      $ 3745 "Loop 1 times"
      Loop_100 = 0
      while (Loop_100 < 1):
        $ 3746 "bajar≔pose_add(get_actual_tcp_pose(), bajada_broca)"
        global bajar= pose_add ( get_actual_tcp_pose (), bajada_broca)
        $ 3747 "bajar" "breakAfter"
        movel(bajar, a=0.005, v=0.001)
        $ 3748 "subir≔pose_sub(get_actual_tcp_pose(), bajada_broca)"
        global subir= pose_sub ( get_actual_tcp_pose (), bajada_broca)
        $ 3749 "subir" "breakAfter"
        movel(subir, a=0.01, v=0.01)
        $ 3750 "bajada_broca≔pose_sub(bajada_broca, bajada)"
        global bajada_broca= pose_sub (bajada_broca, bajada)
        Loop_100 = Loop_100 + 1
      end
      $ 3751 "Direction: Base Z+"
      global move_thread_flag_3751=0
      thread move_thread_3751():
        enter_critical
        move_thread_flag_3751 = 1
        local towardsPos=calculate_point_to_move_towards(p[0.0,0.0,0.0,0.0,0.0,0.0], [0.0,0.0,1.0], 0.06)
        movel(towardsPos, a=0.035, v=0.03)
        move_thread_flag_3751 = 2
        exit_critical
      end
      move_thread_flag_3751 = 0
      move_thread_han_3751 = run move_thread_3751()
      while (True):
        sleep(1.0E-10)
        if (move_thread_flag_3751 > 1):
          join move_thread_han_3751
          $ 3752 "Until (distance)"
          break
        end
        sync()
      end
      $ 3753 "Set CO[1]=Apagar"
      set_configurable_digital_out(1, False)
      $ 3754 "barreno_actual≔barreno_actual+1"
      global barreno_actual=barreno_actual+1
      $ 3755 "Call Quitar_broca"
      Quitar_broca()
      $ 3756 "Call Poner_broca"
      Poner_broca()
    end
    $ 3757 "Popup: Linea3 con full Terminada!"
    popup("Linea3 con full Terminada!", "Mensaje", False, False, blocking=True)
    $ 3758 "Linea4"
    $ 3759 "Marcar_puntos"
    $ 3760 "MoveL"
    $ 3761 "Home3" "breakAfter"
    movel(Home3_p, a=0.5, v=0.1)
    $ 3762 "Linea4_A" "breakAfter"
    movel(Linea4_A_p, a=0.5, v=0.1)
    $ 3763 "Linea4_B" "breakAfter"
    movel(Linea4_B_p, a=0.5, v=0.1)
    $ 3764 "Linea4_C" "breakAfter"
    movel(Linea4_C_p, a=0.5, v=0.1)
    $ 3765 "Linea4_D" "breakAfter"
    movel(Linea4_D_p, a=0.5, v=0.1)
    $ 3766 "Linea4_E" "breakAfter"
    movel(Linea4_E_p, a=0.5, v=0.1)
    $ 3767 "Linea4_F" "breakAfter"
    movel(Linea4_F_p, a=0.5, v=0.1)
    $ 3768 "AB"
    $ 3769 "'desbaste_inicial'"
    # 'desbaste_inicial'
    $ 3770 "bajada_broca≔p[0,0,-0.024,0,0,0]"
    global bajada_broca=p[0,0,-0.024,0,0,0]
    $ 3771 "barrenos_menos1≔8"
    global barrenos_menos1=8
    $ 3772 "barreno_actual≔0"
    global barreno_actual=0
    $ 3773 "Loop barreno_actual≤barrenos_menos1"
    while (barreno_actual <= barrenos_menos1):
      $ 3774 "Perforacion"
      $ 3775 "MoveL"
      $ 3776 "internos≔interpolate_pose(Linea4_A, Linea4_B, barreno_actual/barrenos_menos1)"
      global internos= interpolate_pose (Linea4_A_p, Linea4_B_p, barreno_actual/barrenos_menos1)
      $ 3777 "internos" "breakAfter"
      movel(internos, a=0.5, v=0.1)
      $ 3778 "'desbaste_inicial'"
      # 'desbaste_inicial'
      $ 3779 "bajada_broca≔p[0,0,-0.024,0,0,0]"
      global bajada_broca=p[0,0,-0.024,0,0,0]
      $ 3780 "bajada≔p[0,0,0.024,0,0,0]"
      global bajada=p[0,0,0.024,0,0,0]
      $ 3781 "Direction: Base Z-"
      global move_thread_flag_3781=0
      thread move_thread_3781():
        enter_critical
        move_thread_flag_3781 = 1
        local towardsPos=calculate_point_to_move_towards(p[0.0,0.0,0.0,0.0,0.0,0.0], [0.0,0.0,-1.0], 0.083)
        movel(towardsPos, a=0.035, v=0.03)
        move_thread_flag_3781 = 2
        exit_critical
      end
      move_thread_flag_3781 = 0
      move_thread_han_3781 = run move_thread_3781()
      while (True):
        sleep(1.0E-10)
        if (move_thread_flag_3781 > 1):
          join move_thread_han_3781
          $ 3782 "Until (distance)"
          break
        end
        sync()
      end
      $ 3783 "Popup: punto contacto alanzdo"
      popup("punto contacto alanzdo", "Mensaje", False, False, blocking=True)
      $ 3784 "Direction: Base Z+"
      global move_thread_flag_3784=0
      thread move_thread_3784():
        enter_critical
        move_thread_flag_3784 = 1
        local towardsPos=calculate_point_to_move_towards(p[0.0,0.0,0.0,0.0,0.0,0.0], [0.0,0.0,1.0], 0.002)
        movel(towardsPos, a=0.005, v=0.003)
        move_thread_flag_3784 = 2
        exit_critical
      end
      move_thread_flag_3784 = 0
      move_thread_han_3784 = run move_thread_3784()
      while (True):
        sleep(1.0E-10)
        if (move_thread_flag_3784 > 1):
          join move_thread_han_3784
          $ 3785 "Until (distance)"
          break
        end
        sync()
      end
      $ 3786 "Wait: 0.3"
      sleep(0.3)
      $ 3787 "Set CO[1]=Encender"
      set_configurable_digital_out(1, True)
      $ 3788 "Wait: 0.3"
      sleep(0.3)
      $ 3789 "Loop 1 times"
      Loop_120 = 0
      while (Loop_120 < 1):
        $ 3790 "bajar≔pose_add(get_actual_tcp_pose(), bajada_broca)"
        global bajar= pose_add ( get_actual_tcp_pose (), bajada_broca)
        $ 3791 "bajar" "breakAfter"
        movel(bajar, a=0.005, v=0.001)
        $ 3792 "subir≔pose_sub(get_actual_tcp_pose(), bajada_broca)"
        global subir= pose_sub ( get_actual_tcp_pose (), bajada_broca)
        $ 3793 "subir" "breakAfter"
        movel(subir, a=0.01, v=0.01)
        $ 3794 "bajada_broca≔pose_sub(bajada_broca, bajada)"
        global bajada_broca= pose_sub (bajada_broca, bajada)
        Loop_120 = Loop_120 + 1
      end
      $ 3795 "Direction: Base Z+"
      global move_thread_flag_3795=0
      thread move_thread_3795():
        enter_critical
        move_thread_flag_3795 = 1
        local towardsPos=calculate_point_to_move_towards(p[0.0,0.0,0.0,0.0,0.0,0.0], [0.0,0.0,1.0], 0.06)
        movel(towardsPos, a=0.035, v=0.03)
        move_thread_flag_3795 = 2
        exit_critical
      end
      move_thread_flag_3795 = 0
      move_thread_han_3795 = run move_thread_3795()
      while (True):
        sleep(1.0E-10)
        if (move_thread_flag_3795 > 1):
          join move_thread_han_3795
          $ 3796 "Until (distance)"
          break
        end
        sync()
      end
      $ 3797 "Set CO[1]=Apagar"
      set_configurable_digital_out(1, False)
      $ 3798 "barreno_actual≔barreno_actual+1"
      global barreno_actual=barreno_actual+1
      $ 3799 "Call Quitar_broca"
      Quitar_broca()
      $ 3800 "Call Poner_broca"
      Poner_broca()
    end
    $ 3801 "CD"
    $ 3802 "'desbaste_inicial'"
    # 'desbaste_inicial'
    $ 3803 "bajada_broca≔p[0,0,-0.024,0,0,0]"
    global bajada_broca=p[0,0,-0.024,0,0,0]
    $ 3804 "barrenos_menos1≔8"
    global barrenos_menos1=8
    $ 3805 "barreno_actual≔0"
    global barreno_actual=0
    $ 3806 "Loop barreno_actual≤barrenos_menos1"
    while (barreno_actual <= barrenos_menos1):
      $ 3807 "Perforacion"
      $ 3808 "MoveL"
      $ 3809 "internos≔interpolate_pose(Linea4_C, Linea4_D, barreno_actual/barrenos_menos1)"
      global internos= interpolate_pose (Linea4_C_p, Linea4_D_p, barreno_actual/barrenos_menos1)
      $ 3810 "internos" "breakAfter"
      movel(internos, a=0.5, v=0.1)
      $ 3811 "'desbaste_inicial'"
      # 'desbaste_inicial'
      $ 3812 "bajada_broca≔p[0,0,-0.024,0,0,0]"
      global bajada_broca=p[0,0,-0.024,0,0,0]
      $ 3813 "bajada≔p[0,0,0.024,0,0,0]"
      global bajada=p[0,0,0.024,0,0,0]
      $ 3814 "Direction: Base Z-"
      global move_thread_flag_3814=0
      thread move_thread_3814():
        enter_critical
        move_thread_flag_3814 = 1
        local towardsPos=calculate_point_to_move_towards(p[0.0,0.0,0.0,0.0,0.0,0.0], [0.0,0.0,-1.0], 0.083)
        movel(towardsPos, a=0.035, v=0.03)
        move_thread_flag_3814 = 2
        exit_critical
      end
      move_thread_flag_3814 = 0
      move_thread_han_3814 = run move_thread_3814()
      while (True):
        sleep(1.0E-10)
        if (move_thread_flag_3814 > 1):
          join move_thread_han_3814
          $ 3815 "Until (distance)"
          break
        end
        sync()
      end
      $ 3816 "Popup: punto contacto alanzdo"
      popup("punto contacto alanzdo", "Mensaje", False, False, blocking=True)
      $ 3817 "Direction: Base Z+"
      global move_thread_flag_3817=0
      thread move_thread_3817():
        enter_critical
        move_thread_flag_3817 = 1
        local towardsPos=calculate_point_to_move_towards(p[0.0,0.0,0.0,0.0,0.0,0.0], [0.0,0.0,1.0], 0.002)
        movel(towardsPos, a=0.005, v=0.003)
        move_thread_flag_3817 = 2
        exit_critical
      end
      move_thread_flag_3817 = 0
      move_thread_han_3817 = run move_thread_3817()
      while (True):
        sleep(1.0E-10)
        if (move_thread_flag_3817 > 1):
          join move_thread_han_3817
          $ 3818 "Until (distance)"
          break
        end
        sync()
      end
      $ 3819 "Wait: 0.3"
      sleep(0.3)
      $ 3820 "Set CO[1]=Encender"
      set_configurable_digital_out(1, True)
      $ 3821 "Wait: 0.3"
      sleep(0.3)
      $ 3822 "Loop 1 times"
      Loop_123 = 0
      while (Loop_123 < 1):
        $ 3823 "bajar≔pose_add(get_actual_tcp_pose(), bajada_broca)"
        global bajar= pose_add ( get_actual_tcp_pose (), bajada_broca)
        $ 3824 "bajar" "breakAfter"
        movel(bajar, a=0.005, v=0.001)
        $ 3825 "subir≔pose_sub(get_actual_tcp_pose(), bajada_broca)"
        global subir= pose_sub ( get_actual_tcp_pose (), bajada_broca)
        $ 3826 "subir" "breakAfter"
        movel(subir, a=0.01, v=0.01)
        $ 3827 "bajada_broca≔pose_sub(bajada_broca, bajada)"
        global bajada_broca= pose_sub (bajada_broca, bajada)
        Loop_123 = Loop_123 + 1
      end
      $ 3828 "Direction: Base Z+"
      global move_thread_flag_3828=0
      thread move_thread_3828():
        enter_critical
        move_thread_flag_3828 = 1
        local towardsPos=calculate_point_to_move_towards(p[0.0,0.0,0.0,0.0,0.0,0.0], [0.0,0.0,1.0], 0.06)
        movel(towardsPos, a=0.035, v=0.03)
        move_thread_flag_3828 = 2
        exit_critical
      end
      move_thread_flag_3828 = 0
      move_thread_han_3828 = run move_thread_3828()
      while (True):
        sleep(1.0E-10)
        if (move_thread_flag_3828 > 1):
          join move_thread_han_3828
          $ 3829 "Until (distance)"
          break
        end
        sync()
      end
      $ 3830 "Set CO[1]=Apagar"
      set_configurable_digital_out(1, False)
      $ 3831 "barreno_actual≔barreno_actual+1"
      global barreno_actual=barreno_actual+1
      $ 3832 "Call Quitar_broca"
      Quitar_broca()
      $ 3833 "Call Poner_broca"
      Poner_broca()
    end
    $ 3834 "EF"
    $ 3835 "'desbaste_inicial'"
    # 'desbaste_inicial'
    $ 3836 "bajada_broca≔p[0,0,-0.024,0,0,0]"
    global bajada_broca=p[0,0,-0.024,0,0,0]
    $ 3837 "barrenos_menos1≔8"
    global barrenos_menos1=8
    $ 3838 "barreno_actual≔0"
    global barreno_actual=0
    $ 3839 "Loop barreno_actual≤barrenos_menos1"
    while (barreno_actual <= barrenos_menos1):
      $ 3840 "Perforacion"
      $ 3841 "MoveL"
      $ 3842 "internos≔interpolate_pose(Linea4_E, Linea4_F, barreno_actual/barrenos_menos1)"
      global internos= interpolate_pose (Linea4_E_p, Linea4_F_p, barreno_actual/barrenos_menos1)
      $ 3843 "internos" "breakAfter"
      movel(internos, a=0.5, v=0.1)
      $ 3844 "'desbaste_inicial'"
      # 'desbaste_inicial'
      $ 3845 "bajada_broca≔p[0,0,-0.024,0,0,0]"
      global bajada_broca=p[0,0,-0.024,0,0,0]
      $ 3846 "bajada≔p[0,0,0.024,0,0,0]"
      global bajada=p[0,0,0.024,0,0,0]
      $ 3847 "Direction: Base Z-"
      global move_thread_flag_3847=0
      thread move_thread_3847():
        enter_critical
        move_thread_flag_3847 = 1
        local towardsPos=calculate_point_to_move_towards(p[0.0,0.0,0.0,0.0,0.0,0.0], [0.0,0.0,-1.0], 0.083)
        movel(towardsPos, a=0.035, v=0.03)
        move_thread_flag_3847 = 2
        exit_critical
      end
      move_thread_flag_3847 = 0
      move_thread_han_3847 = run move_thread_3847()
      while (True):
        sleep(1.0E-10)
        if (move_thread_flag_3847 > 1):
          join move_thread_han_3847
          $ 3848 "Until (distance)"
          break
        end
        sync()
      end
      $ 3849 "Popup: punto contacto alanzdo"
      popup("punto contacto alanzdo", "Mensaje", False, False, blocking=True)
      $ 3850 "Direction: Base Z+"
      global move_thread_flag_3850=0
      thread move_thread_3850():
        enter_critical
        move_thread_flag_3850 = 1
        local towardsPos=calculate_point_to_move_towards(p[0.0,0.0,0.0,0.0,0.0,0.0], [0.0,0.0,1.0], 0.002)
        movel(towardsPos, a=0.005, v=0.003)
        move_thread_flag_3850 = 2
        exit_critical
      end
      move_thread_flag_3850 = 0
      move_thread_han_3850 = run move_thread_3850()
      while (True):
        sleep(1.0E-10)
        if (move_thread_flag_3850 > 1):
          join move_thread_han_3850
          $ 3851 "Until (distance)"
          break
        end
        sync()
      end
      $ 3852 "Wait: 0.3"
      sleep(0.3)
      $ 3853 "Set CO[1]=Encender"
      set_configurable_digital_out(1, True)
      $ 3854 "Wait: 0.3"
      sleep(0.3)
      $ 3855 "Loop 1 times"
      Loop_125 = 0
      while (Loop_125 < 1):
        $ 3856 "bajar≔pose_add(get_actual_tcp_pose(), bajada_broca)"
        global bajar= pose_add ( get_actual_tcp_pose (), bajada_broca)
        $ 3857 "bajar" "breakAfter"
        movel(bajar, a=0.005, v=0.001)
        $ 3858 "subir≔pose_sub(get_actual_tcp_pose(), bajada_broca)"
        global subir= pose_sub ( get_actual_tcp_pose (), bajada_broca)
        $ 3859 "subir" "breakAfter"
        movel(subir, a=0.01, v=0.01)
        $ 3860 "bajada_broca≔pose_sub(bajada_broca, bajada)"
        global bajada_broca= pose_sub (bajada_broca, bajada)
        Loop_125 = Loop_125 + 1
      end
      $ 3861 "Direction: Base Z+"
      global move_thread_flag_3861=0
      thread move_thread_3861():
        enter_critical
        move_thread_flag_3861 = 1
        local towardsPos=calculate_point_to_move_towards(p[0.0,0.0,0.0,0.0,0.0,0.0], [0.0,0.0,1.0], 0.06)
        movel(towardsPos, a=0.035, v=0.03)
        move_thread_flag_3861 = 2
        exit_critical
      end
      move_thread_flag_3861 = 0
      move_thread_han_3861 = run move_thread_3861()
      while (True):
        sleep(1.0E-10)
        if (move_thread_flag_3861 > 1):
          join move_thread_han_3861
          $ 3862 "Until (distance)"
          break
        end
        sync()
      end
      $ 3863 "Set CO[1]=Apagar"
      set_configurable_digital_out(1, False)
      $ 3864 "barreno_actual≔barreno_actual+1"
      global barreno_actual=barreno_actual+1
      $ 3865 "If barreno_actual>barrenos_menos1"
      if (barreno_actual>barrenos_menos1):
        $ 3866 "cambiar_broca≔ True "
        global cambiar_broca=  True
      end
      $ 3867 "Call Quitar_broca"
      Quitar_broca()
      $ 3868 "Call Poner_broca"
      Poner_broca()
    end
    $ 3869 "Popup: Linea4 con full Terminada!"
    popup("Linea4 con full Terminada!", "Mensaje", False, False, blocking=True)
    $ 4090 "720"
    $ 4091 "Broca_1"
    $ 4092 "Linea19"
    $ 4093 "Marcar_puntos"
    $ 4094 "MoveL"
    $ 4095 "Home3" "breakAfter"
    movel(Home3_p, a=0.5, v=0.1)
    $ 4096 "Linea19_A" "breakAfter"
    movel(Linea19_A_p, a=0.5, v=0.1)
    $ 4097 "bajada_comprobacion"
    $ 4098 "Direction: Base Z-"
    global move_thread_flag_4098=0
    thread move_thread_4098():
      enter_critical
      move_thread_flag_4098 = 1
      local towardsPos=calculate_point_to_move_towards(p[0.0,0.0,0.0,0.0,0.0,0.0], [0.0,0.0,-1.0], 0.071)
      movel(towardsPos, a=0.15, v=0.1)
      move_thread_flag_4098 = 2
      exit_critical
    end
    move_thread_flag_4098 = 0
    move_thread_han_4098 = run move_thread_4098()
    while (True):
      sleep(1.0E-10)
      if (move_thread_flag_4098 > 1):
        join move_thread_han_4098
        $ 4099 "Until (distance)"
        break
      end
      sync()
    end
    $ 4100 "Direction: Base Z-"
    global move_thread_flag_4100=0
    thread move_thread_4100():
      enter_critical
      move_thread_flag_4100 = 1
      local towardsPos=calculate_point_to_move_towards(p[0.0,0.0,0.0,0.0,0.0,0.0], [0.0,0.0,-1.0], 1000.0)
      movel(towardsPos, a=0.007, v=0.007)
      move_thread_flag_4100 = 2
      exit_critical
    end
    move_thread_flag_4100 = 0
    move_thread_han_4100 = run move_thread_4100()
    while (True):
      local targetTcpDirection=get_target_tcp_speed()
      local stepsToRetract=tool_contact(direction=targetTcpDirection)
      if (stepsToRetract > 0):
        kill move_thread_han_4100
        stopl(0.02)
        local backTrackMovement=get_actual_joint_positions_history(stepsToRetract)
        local contactPose=get_forward_kin(backTrackMovement)
        local posDir=[targetTcpDirection[0],targetTcpDirection[1],targetTcpDirection[2]]
        local retractTo=contactPose
        if (norm(posDir) > 1e-6):
          local normalizedPosDir=normalize(posDir)
          local additionalRetraction=p[normalizedPosDir[0] * 0.0, normalizedPosDir[1] * 0.0, normalizedPosDir[2] * 0.0, 0, 0, 0]
          retractTo = pose_sub(contactPose, additionalRetraction)
        end
        movel(retractTo, a=0.02, v=0.1)
        $ 4101 "Until (tool_contact_detection)"
        break
      end
      sync()
    end
    $ 4102 "Direction: Base Z+"
    global move_thread_flag_4102=0
    thread move_thread_4102():
      enter_critical
      move_thread_flag_4102 = 1
      local towardsPos=calculate_point_to_move_towards(p[0.0,0.0,0.0,0.0,0.0,0.0], [0.0,0.0,1.0], 0.08)
      movel(towardsPos, a=0.15, v=0.1)
      move_thread_flag_4102 = 2
      exit_critical
    end
    move_thread_flag_4102 = 0
    move_thread_han_4102 = run move_thread_4102()
    while (True):
      sleep(1.0E-10)
      if (move_thread_flag_4102 > 1):
        join move_thread_han_4102
        $ 4103 "Until (distance)"
        break
      end
      sync()
    end
    $ 4104 "Linea19_B" "breakAfter"
    movel(Linea19_B_p, a=0.5, v=0.1)
    $ 4105 "bajada_comprobacion"
    $ 4106 "Direction: Base Z-"
    global move_thread_flag_4106=0
    thread move_thread_4106():
      enter_critical
      move_thread_flag_4106 = 1
      local towardsPos=calculate_point_to_move_towards(p[0.0,0.0,0.0,0.0,0.0,0.0], [0.0,0.0,-1.0], 0.071)
      movel(towardsPos, a=0.15, v=0.1)
      move_thread_flag_4106 = 2
      exit_critical
    end
    move_thread_flag_4106 = 0
    move_thread_han_4106 = run move_thread_4106()
    while (True):
      sleep(1.0E-10)
      if (move_thread_flag_4106 > 1):
        join move_thread_han_4106
        $ 4107 "Until (distance)"
        break
      end
      sync()
    end
    $ 4108 "Direction: Base Z-"
    global move_thread_flag_4108=0
    thread move_thread_4108():
      enter_critical
      move_thread_flag_4108 = 1
      local towardsPos=calculate_point_to_move_towards(p[0.0,0.0,0.0,0.0,0.0,0.0], [0.0,0.0,-1.0], 1000.0)
      movel(towardsPos, a=0.007, v=0.007)
      move_thread_flag_4108 = 2
      exit_critical
    end
    move_thread_flag_4108 = 0
    move_thread_han_4108 = run move_thread_4108()
    while (True):
      local targetTcpDirection=get_target_tcp_speed()
      local stepsToRetract=tool_contact(direction=targetTcpDirection)
      if (stepsToRetract > 0):
        kill move_thread_han_4108
        stopl(0.02)
        local backTrackMovement=get_actual_joint_positions_history(stepsToRetract)
        local contactPose=get_forward_kin(backTrackMovement)
        local posDir=[targetTcpDirection[0],targetTcpDirection[1],targetTcpDirection[2]]
        local retractTo=contactPose
        if (norm(posDir) > 1e-6):
          local normalizedPosDir=normalize(posDir)
          local additionalRetraction=p[normalizedPosDir[0] * 0.0, normalizedPosDir[1] * 0.0, normalizedPosDir[2] * 0.0, 0, 0, 0]
          retractTo = pose_sub(contactPose, additionalRetraction)
        end
        movel(retractTo, a=0.02, v=0.1)
        $ 4109 "Until (tool_contact_detection)"
        break
      end
      sync()
    end
    $ 4110 "Direction: Base Z+"
    global move_thread_flag_4110=0
    thread move_thread_4110():
      enter_critical
      move_thread_flag_4110 = 1
      local towardsPos=calculate_point_to_move_towards(p[0.0,0.0,0.0,0.0,0.0,0.0], [0.0,0.0,1.0], 0.08)
      movel(towardsPos, a=0.15, v=0.1)
      move_thread_flag_4110 = 2
      exit_critical
    end
    move_thread_flag_4110 = 0
    move_thread_han_4110 = run move_thread_4110()
    while (True):
      sleep(1.0E-10)
      if (move_thread_flag_4110 > 1):
        join move_thread_han_4110
        $ 4111 "Until (distance)"
        break
      end
      sync()
    end
    $ 4112 "AB"
    $ 4113 "'desbaste_inicial'"
    # 'desbaste_inicial'
    $ 4114 "bajada_broca≔p[0,0,-0.008,0,0,0]"
    global bajada_broca=p[0,0,-0.008,0,0,0]
    $ 4115 "barrenos_menos1≔1"
    global barrenos_menos1=1
    $ 4116 "barreno_actual≔0"
    global barreno_actual=0
    $ 4117 "Loop barreno_actual≤barrenos_menos1"
    while (barreno_actual <= barrenos_menos1):
      $ 4118 "Perforacion"
      $ 4119 "MoveL"
      $ 4120 "internos≔interpolate_pose(Linea19_A, Linea19_B, barreno_actual/barrenos_menos1)"
      global internos= interpolate_pose (Linea19_A_p, Linea19_B_p, barreno_actual/barrenos_menos1)
      $ 4121 "internos" "breakAfter"
      movel(internos, a=0.5, v=0.1)
      $ 4122 "'desbaste_inicial'"
      # 'desbaste_inicial'
      $ 4123 "bajada_broca≔p[0,0,-0.024,0,0,0]"
      global bajada_broca=p[0,0,-0.024,0,0,0]
      $ 4124 "bajada≔p[0,0,0.024,0,0,0]"
      global bajada=p[0,0,0.024,0,0,0]
      $ 4125 "Direction: Base Z-"
      global move_thread_flag_4125=0
      thread move_thread_4125():
        enter_critical
        move_thread_flag_4125 = 1
        local towardsPos=calculate_point_to_move_towards(p[0.0,0.0,0.0,0.0,0.0,0.0], [0.0,0.0,-1.0], 0.071)
        movel(towardsPos, a=0.15, v=0.1)
        move_thread_flag_4125 = 2
        exit_critical
      end
      move_thread_flag_4125 = 0
      move_thread_han_4125 = run move_thread_4125()
      while (True):
        sleep(1.0E-10)
        if (move_thread_flag_4125 > 1):
          join move_thread_han_4125
          $ 4126 "Until (distance)"
          break
        end
        sync()
      end
      $ 4127 "Direction: Base Z-"
      global move_thread_flag_4127=0
      thread move_thread_4127():
        enter_critical
        move_thread_flag_4127 = 1
        local towardsPos=calculate_point_to_move_towards(p[0.0,0.0,0.0,0.0,0.0,0.0], [0.0,0.0,-1.0], 1000.0)
        movel(towardsPos, a=0.007, v=0.007)
        move_thread_flag_4127 = 2
        exit_critical
      end
      move_thread_flag_4127 = 0
      move_thread_han_4127 = run move_thread_4127()
      while (True):
        local targetTcpDirection=get_target_tcp_speed()
        local stepsToRetract=tool_contact(direction=targetTcpDirection)
        if (stepsToRetract > 0):
          kill move_thread_han_4127
          stopl(0.02)
          local backTrackMovement=get_actual_joint_positions_history(stepsToRetract)
          local contactPose=get_forward_kin(backTrackMovement)
          local posDir=[targetTcpDirection[0],targetTcpDirection[1],targetTcpDirection[2]]
          local retractTo=contactPose
          if (norm(posDir) > 1e-6):
            local normalizedPosDir=normalize(posDir)
            local additionalRetraction=p[normalizedPosDir[0] * 0.0, normalizedPosDir[1] * 0.0, normalizedPosDir[2] * 0.0, 0, 0, 0]
            retractTo = pose_sub(contactPose, additionalRetraction)
          end
          movel(retractTo, a=0.02, v=0.1)
          $ 4128 "Until (tool_contact_detection)"
          break
        end
        sync()
      end
      $ 4129 "Popup: punto contacto alanzdo"
      popup("punto contacto alanzdo", "Mensaje", False, False, blocking=True)
      $ 4130 "Direction: Base Z+"
      global move_thread_flag_4130=0
      thread move_thread_4130():
        enter_critical
        move_thread_flag_4130 = 1
        local towardsPos=calculate_point_to_move_towards(p[0.0,0.0,0.0,0.0,0.0,0.0], [0.0,0.0,1.0], 0.007)
        movel(towardsPos, a=0.015, v=0.015)
        move_thread_flag_4130 = 2
        exit_critical
      end
      move_thread_flag_4130 = 0
      move_thread_han_4130 = run move_thread_4130()
      while (True):
        sleep(1.0E-10)
        if (move_thread_flag_4130 > 1):
          join move_thread_han_4130
          $ 4131 "Until (distance)"
          break
        end
        sync()
      end
      $ 4132 "Wait: 0.3"
      sleep(0.3)
      $ 4133 "Set CO[1]=Encender"
      set_configurable_digital_out(1, True)
      $ 4134 "Wait: 0.3"
      sleep(0.3)
      $ 4135 "Loop 1 times"
      Loop_47 = 0
      while (Loop_47 < 1):
        $ 4136 "bajar≔pose_add(get_actual_tcp_pose(), bajada_broca)"
        global bajar= pose_add ( get_actual_tcp_pose (), bajada_broca)
        $ 4137 "bajar" "breakAfter"
        movel(bajar, a=0.004, v=0.004)
        $ 4138 "subir≔pose_sub(get_actual_tcp_pose(), bajada_broca)"
        global subir= pose_sub ( get_actual_tcp_pose (), bajada_broca)
        $ 4139 "Direction: Base Z+"
        global move_thread_flag_4139=0
        thread move_thread_4139():
          enter_critical
          move_thread_flag_4139 = 1
          local towardsPos=calculate_point_to_move_towards(p[0.0,0.0,0.0,0.0,0.0,0.0], [0.0,0.0,1.0], 0.002)
          movel(towardsPos, a=0.015, v=0.015)
          move_thread_flag_4139 = 2
          exit_critical
        end
        move_thread_flag_4139 = 0
        move_thread_han_4139 = run move_thread_4139()
        while (True):
          sleep(1.0E-10)
          if (move_thread_flag_4139 > 1):
            join move_thread_han_4139
            $ 4140 "Until (distance)"
            break
          end
          sync()
        end
        $ 4141 "Set CO[1]=Apagar"
        set_configurable_digital_out(1, False)
        $ 4142 "subir" "breakAfter"
        movel(subir, a=0.015, v=0.015)
        $ 4143 "bajada_broca≔pose_sub(bajada_broca, bajada)"
        global bajada_broca= pose_sub (bajada_broca, bajada)
        Loop_47 = Loop_47 + 1
      end
      $ 4144 "Direction: Base Z+"
      global move_thread_flag_4144=0
      thread move_thread_4144():
        enter_critical
        move_thread_flag_4144 = 1
        local towardsPos=calculate_point_to_move_towards(p[0.0,0.0,0.0,0.0,0.0,0.0], [0.0,0.0,1.0], 0.08)
        movel(towardsPos, a=0.15, v=0.1)
        move_thread_flag_4144 = 2
        exit_critical
      end
      move_thread_flag_4144 = 0
      move_thread_han_4144 = run move_thread_4144()
      while (True):
        sleep(1.0E-10)
        if (move_thread_flag_4144 > 1):
          join move_thread_han_4144
          $ 4145 "Until (distance)"
          break
        end
        sync()
      end
      $ 4146 "Set CO[1]=Apagar"
      set_configurable_digital_out(1, False)
      $ 4147 "barreno_actual≔barreno_actual+1"
      global barreno_actual=barreno_actual+1
    end
    $ 4150 "Popup: Linea19 con chica Terminada!"
    popup("Linea19 con chica Terminada!", "Mensaje", False, False, blocking=True)
    $ 4151 "Linea20"
    $ 4152 "Marcar_puntos"
    $ 4153 "MoveL"
    $ 4154 "Linea20_A" "breakAfter"
    movel(Linea20_A_p, a=0.5, v=0.1)
    $ 4155 "bajada_comprobacion"
    $ 4156 "Direction: Base Z-"
    global move_thread_flag_4156=0
    thread move_thread_4156():
      enter_critical
      move_thread_flag_4156 = 1
      local towardsPos=calculate_point_to_move_towards(p[0.0,0.0,0.0,0.0,0.0,0.0], [0.0,0.0,-1.0], 0.071)
      movel(towardsPos, a=0.15, v=0.1)
      move_thread_flag_4156 = 2
      exit_critical
    end
    move_thread_flag_4156 = 0
    move_thread_han_4156 = run move_thread_4156()
    while (True):
      sleep(1.0E-10)
      if (move_thread_flag_4156 > 1):
        join move_thread_han_4156
        $ 4157 "Until (distance)"
        break
      end
      sync()
    end
    $ 4158 "Direction: Base Z-"
    global move_thread_flag_4158=0
    thread move_thread_4158():
      enter_critical
      move_thread_flag_4158 = 1
      local towardsPos=calculate_point_to_move_towards(p[0.0,0.0,0.0,0.0,0.0,0.0], [0.0,0.0,-1.0], 1000.0)
      movel(towardsPos, a=0.007, v=0.007)
      move_thread_flag_4158 = 2
      exit_critical
    end
    move_thread_flag_4158 = 0
    move_thread_han_4158 = run move_thread_4158()
    while (True):
      local targetTcpDirection=get_target_tcp_speed()
      local stepsToRetract=tool_contact(direction=targetTcpDirection)
      if (stepsToRetract > 0):
        kill move_thread_han_4158
        stopl(0.02)
        local backTrackMovement=get_actual_joint_positions_history(stepsToRetract)
        local contactPose=get_forward_kin(backTrackMovement)
        local posDir=[targetTcpDirection[0],targetTcpDirection[1],targetTcpDirection[2]]
        local retractTo=contactPose
        if (norm(posDir) > 1e-6):
          local normalizedPosDir=normalize(posDir)
          local additionalRetraction=p[normalizedPosDir[0] * 0.0, normalizedPosDir[1] * 0.0, normalizedPosDir[2] * 0.0, 0, 0, 0]
          retractTo = pose_sub(contactPose, additionalRetraction)
        end
        movel(retractTo, a=0.02, v=0.1)
        $ 4159 "Until (tool_contact_detection)"
        break
      end
      sync()
    end
    $ 4160 "Direction: Base Z+"
    global move_thread_flag_4160=0
    thread move_thread_4160():
      enter_critical
      move_thread_flag_4160 = 1
      local towardsPos=calculate_point_to_move_towards(p[0.0,0.0,0.0,0.0,0.0,0.0], [0.0,0.0,1.0], 0.08)
      movel(towardsPos, a=0.15, v=0.1)
      move_thread_flag_4160 = 2
      exit_critical
    end
    move_thread_flag_4160 = 0
    move_thread_han_4160 = run move_thread_4160()
    while (True):
      sleep(1.0E-10)
      if (move_thread_flag_4160 > 1):
        join move_thread_han_4160
        $ 4161 "Until (distance)"
        break
      end
      sync()
    end
    $ 4162 "Linea20_B" "breakAfter"
    movel(Linea20_B_p, a=0.5, v=0.1)
    $ 4163 "bajada_comprobacion"
    $ 4164 "Direction: Base Z-"
    global move_thread_flag_4164=0
    thread move_thread_4164():
      enter_critical
      move_thread_flag_4164 = 1
      local towardsPos=calculate_point_to_move_towards(p[0.0,0.0,0.0,0.0,0.0,0.0], [0.0,0.0,-1.0], 0.071)
      movel(towardsPos, a=0.15, v=0.1)
      move_thread_flag_4164 = 2
      exit_critical
    end
    move_thread_flag_4164 = 0
    move_thread_han_4164 = run move_thread_4164()
    while (True):
      sleep(1.0E-10)
      if (move_thread_flag_4164 > 1):
        join move_thread_han_4164
        $ 4165 "Until (distance)"
        break
      end
      sync()
    end
    $ 4166 "Direction: Base Z-"
    global move_thread_flag_4166=0
    thread move_thread_4166():
      enter_critical
      move_thread_flag_4166 = 1
      local towardsPos=calculate_point_to_move_towards(p[0.0,0.0,0.0,0.0,0.0,0.0], [0.0,0.0,-1.0], 1000.0)
      movel(towardsPos, a=0.007, v=0.007)
      move_thread_flag_4166 = 2
      exit_critical
    end
    move_thread_flag_4166 = 0
    move_thread_han_4166 = run move_thread_4166()
    while (True):
      local targetTcpDirection=get_target_tcp_speed()
      local stepsToRetract=tool_contact(direction=targetTcpDirection)
      if (stepsToRetract > 0):
        kill move_thread_han_4166
        stopl(0.02)
        local backTrackMovement=get_actual_joint_positions_history(stepsToRetract)
        local contactPose=get_forward_kin(backTrackMovement)
        local posDir=[targetTcpDirection[0],targetTcpDirection[1],targetTcpDirection[2]]
        local retractTo=contactPose
        if (norm(posDir) > 1e-6):
          local normalizedPosDir=normalize(posDir)
          local additionalRetraction=p[normalizedPosDir[0] * 0.0, normalizedPosDir[1] * 0.0, normalizedPosDir[2] * 0.0, 0, 0, 0]
          retractTo = pose_sub(contactPose, additionalRetraction)
        end
        movel(retractTo, a=0.02, v=0.1)
        $ 4167 "Until (tool_contact_detection)"
        break
      end
      sync()
    end
    $ 4168 "Direction: Base Z+"
    global move_thread_flag_4168=0
    thread move_thread_4168():
      enter_critical
      move_thread_flag_4168 = 1
      local towardsPos=calculate_point_to_move_towards(p[0.0,0.0,0.0,0.0,0.0,0.0], [0.0,0.0,1.0], 0.08)
      movel(towardsPos, a=0.15, v=0.1)
      move_thread_flag_4168 = 2
      exit_critical
    end
    move_thread_flag_4168 = 0
    move_thread_han_4168 = run move_thread_4168()
    while (True):
      sleep(1.0E-10)
      if (move_thread_flag_4168 > 1):
        join move_thread_han_4168
        $ 4169 "Until (distance)"
        break
      end
      sync()
    end
    $ 4170 "AB"
    $ 4171 "'desbaste_inicial'"
    # 'desbaste_inicial'
    $ 4172 "bajada_broca≔p[0,0,-0.008,0,0,0]"
    global bajada_broca=p[0,0,-0.008,0,0,0]
    $ 4173 "barrenos_menos1≔2"
    global barrenos_menos1=2
    $ 4174 "barreno_actual≔0"
    global barreno_actual=0
    $ 4175 "Loop barreno_actual≤barrenos_menos1"
    while (barreno_actual <= barrenos_menos1):
      $ 4176 "Perforacion"
      $ 4177 "MoveL"
      $ 4178 "internos≔interpolate_pose(Linea20_A, Linea20_B, barreno_actual/barrenos_menos1)"
      global internos= interpolate_pose (Linea20_A_p, Linea20_B_p, barreno_actual/barrenos_menos1)
      $ 4179 "internos" "breakAfter"
      movel(internos, a=0.5, v=0.1)
      $ 4180 "'desbaste_inicial'"
      # 'desbaste_inicial'
      $ 4181 "bajada_broca≔p[0,0,-0.024,0,0,0]"
      global bajada_broca=p[0,0,-0.024,0,0,0]
      $ 4182 "bajada≔p[0,0,0.024,0,0,0]"
      global bajada=p[0,0,0.024,0,0,0]
      $ 4183 "Direction: Base Z-"
      global move_thread_flag_4183=0
      thread move_thread_4183():
        enter_critical
        move_thread_flag_4183 = 1
        local towardsPos=calculate_point_to_move_towards(p[0.0,0.0,0.0,0.0,0.0,0.0], [0.0,0.0,-1.0], 0.071)
        movel(towardsPos, a=0.15, v=0.1)
        move_thread_flag_4183 = 2
        exit_critical
      end
      move_thread_flag_4183 = 0
      move_thread_han_4183 = run move_thread_4183()
      while (True):
        sleep(1.0E-10)
        if (move_thread_flag_4183 > 1):
          join move_thread_han_4183
          $ 4184 "Until (distance)"
          break
        end
        sync()
      end
      $ 4185 "Direction: Base Z-"
      global move_thread_flag_4185=0
      thread move_thread_4185():
        enter_critical
        move_thread_flag_4185 = 1
        local towardsPos=calculate_point_to_move_towards(p[0.0,0.0,0.0,0.0,0.0,0.0], [0.0,0.0,-1.0], 1000.0)
        movel(towardsPos, a=0.007, v=0.007)
        move_thread_flag_4185 = 2
        exit_critical
      end
      move_thread_flag_4185 = 0
      move_thread_han_4185 = run move_thread_4185()
      while (True):
        local targetTcpDirection=get_target_tcp_speed()
        local stepsToRetract=tool_contact(direction=targetTcpDirection)
        if (stepsToRetract > 0):
          kill move_thread_han_4185
          stopl(0.02)
          local backTrackMovement=get_actual_joint_positions_history(stepsToRetract)
          local contactPose=get_forward_kin(backTrackMovement)
          local posDir=[targetTcpDirection[0],targetTcpDirection[1],targetTcpDirection[2]]
          local retractTo=contactPose
          if (norm(posDir) > 1e-6):
            local normalizedPosDir=normalize(posDir)
            local additionalRetraction=p[normalizedPosDir[0] * 0.0, normalizedPosDir[1] * 0.0, normalizedPosDir[2] * 0.0, 0, 0, 0]
            retractTo = pose_sub(contactPose, additionalRetraction)
          end
          movel(retractTo, a=0.02, v=0.1)
          $ 4186 "Until (tool_contact_detection)"
          break
        end
        sync()
      end
      $ 4187 "Popup: punto contacto alanzdo"
      popup("punto contacto alanzdo", "Mensaje", False, False, blocking=True)
      $ 4188 "Direction: Base Z+"
      global move_thread_flag_4188=0
      thread move_thread_4188():
        enter_critical
        move_thread_flag_4188 = 1
        local towardsPos=calculate_point_to_move_towards(p[0.0,0.0,0.0,0.0,0.0,0.0], [0.0,0.0,1.0], 0.007)
        movel(towardsPos, a=0.015, v=0.015)
        move_thread_flag_4188 = 2
        exit_critical
      end
      move_thread_flag_4188 = 0
      move_thread_han_4188 = run move_thread_4188()
      while (True):
        sleep(1.0E-10)
        if (move_thread_flag_4188 > 1):
          join move_thread_han_4188
          $ 4189 "Until (distance)"
          break
        end
        sync()
      end
      $ 4190 "Wait: 0.3"
      sleep(0.3)
      $ 4191 "Set CO[1]=Encender"
      set_configurable_digital_out(1, True)
      $ 4192 "Wait: 0.3"
      sleep(0.3)
      $ 4193 "Loop 1 times"
      Loop_57 = 0
      while (Loop_57 < 1):
        $ 4194 "bajar≔pose_add(get_actual_tcp_pose(), bajada_broca)"
        global bajar= pose_add ( get_actual_tcp_pose (), bajada_broca)
        $ 4195 "bajar" "breakAfter"
        movel(bajar, a=0.004, v=0.004)
        $ 4196 "subir≔pose_sub(get_actual_tcp_pose(), bajada_broca)"
        global subir= pose_sub ( get_actual_tcp_pose (), bajada_broca)
        $ 4197 "Direction: Base Z+"
        global move_thread_flag_4197=0
        thread move_thread_4197():
          enter_critical
          move_thread_flag_4197 = 1
          local towardsPos=calculate_point_to_move_towards(p[0.0,0.0,0.0,0.0,0.0,0.0], [0.0,0.0,1.0], 0.002)
          movel(towardsPos, a=0.015, v=0.015)
          move_thread_flag_4197 = 2
          exit_critical
        end
        move_thread_flag_4197 = 0
        move_thread_han_4197 = run move_thread_4197()
        while (True):
          sleep(1.0E-10)
          if (move_thread_flag_4197 > 1):
            join move_thread_han_4197
            $ 4198 "Until (distance)"
            break
          end
          sync()
        end
        $ 4199 "Set CO[1]=Apagar"
        set_configurable_digital_out(1, False)
        $ 4200 "subir" "breakAfter"
        movel(subir, a=0.015, v=0.015)
        $ 4201 "bajada_broca≔pose_sub(bajada_broca, bajada)"
        global bajada_broca= pose_sub (bajada_broca, bajada)
        Loop_57 = Loop_57 + 1
      end
      $ 4202 "Direction: Base Z+"
      global move_thread_flag_4202=0
      thread move_thread_4202():
        enter_critical
        move_thread_flag_4202 = 1
        local towardsPos=calculate_point_to_move_towards(p[0.0,0.0,0.0,0.0,0.0,0.0], [0.0,0.0,1.0], 0.08)
        movel(towardsPos, a=0.15, v=0.1)
        move_thread_flag_4202 = 2
        exit_critical
      end
      move_thread_flag_4202 = 0
      move_thread_han_4202 = run move_thread_4202()
      while (True):
        sleep(1.0E-10)
        if (move_thread_flag_4202 > 1):
          join move_thread_han_4202
          $ 4203 "Until (distance)"
          break
        end
        sync()
      end
      $ 4204 "Set CO[1]=Apagar"
      set_configurable_digital_out(1, False)
      $ 4205 "barreno_actual≔barreno_actual+1"
      global barreno_actual=barreno_actual+1
    end
    $ 4208 "Popup: Linea20 con chica Terminada!"
    popup("Linea20 con chica Terminada!", "Mensaje", False, False, blocking=True)
    $ 4209 "Linea21"
    $ 4210 "Marcar_puntos"
    $ 4211 "MoveL"
    $ 4212 "Linea21_A" "breakAfter"
    movel(Linea21_A_p, a=0.5, v=0.1)
    $ 4213 "bajada_comprobacion"
    $ 4214 "Direction: Base Z-"
    global move_thread_flag_4214=0
    thread move_thread_4214():
      enter_critical
      move_thread_flag_4214 = 1
      local towardsPos=calculate_point_to_move_towards(p[0.0,0.0,0.0,0.0,0.0,0.0], [0.0,0.0,-1.0], 0.071)
      movel(towardsPos, a=0.15, v=0.1)
      move_thread_flag_4214 = 2
      exit_critical
    end
    move_thread_flag_4214 = 0
    move_thread_han_4214 = run move_thread_4214()
    while (True):
      sleep(1.0E-10)
      if (move_thread_flag_4214 > 1):
        join move_thread_han_4214
        $ 4215 "Until (distance)"
        break
      end
      sync()
    end
    $ 4216 "Direction: Base Z-"
    global move_thread_flag_4216=0
    thread move_thread_4216():
      enter_critical
      move_thread_flag_4216 = 1
      local towardsPos=calculate_point_to_move_towards(p[0.0,0.0,0.0,0.0,0.0,0.0], [0.0,0.0,-1.0], 1000.0)
      movel(towardsPos, a=0.007, v=0.007)
      move_thread_flag_4216 = 2
      exit_critical
    end
    move_thread_flag_4216 = 0
    move_thread_han_4216 = run move_thread_4216()
    while (True):
      local targetTcpDirection=get_target_tcp_speed()
      local stepsToRetract=tool_contact(direction=targetTcpDirection)
      if (stepsToRetract > 0):
        kill move_thread_han_4216
        stopl(0.02)
        local backTrackMovement=get_actual_joint_positions_history(stepsToRetract)
        local contactPose=get_forward_kin(backTrackMovement)
        local posDir=[targetTcpDirection[0],targetTcpDirection[1],targetTcpDirection[2]]
        local retractTo=contactPose
        if (norm(posDir) > 1e-6):
          local normalizedPosDir=normalize(posDir)
          local additionalRetraction=p[normalizedPosDir[0] * 0.0, normalizedPosDir[1] * 0.0, normalizedPosDir[2] * 0.0, 0, 0, 0]
          retractTo = pose_sub(contactPose, additionalRetraction)
        end
        movel(retractTo, a=0.02, v=0.1)
        $ 4217 "Until (tool_contact_detection)"
        break
      end
      sync()
    end
    $ 4218 "Direction: Base Z+"
    global move_thread_flag_4218=0
    thread move_thread_4218():
      enter_critical
      move_thread_flag_4218 = 1
      local towardsPos=calculate_point_to_move_towards(p[0.0,0.0,0.0,0.0,0.0,0.0], [0.0,0.0,1.0], 0.08)
      movel(towardsPos, a=0.15, v=0.1)
      move_thread_flag_4218 = 2
      exit_critical
    end
    move_thread_flag_4218 = 0
    move_thread_han_4218 = run move_thread_4218()
    while (True):
      sleep(1.0E-10)
      if (move_thread_flag_4218 > 1):
        join move_thread_han_4218
        $ 4219 "Until (distance)"
        break
      end
      sync()
    end
    $ 4221 "Linea21_AB" "breakAfter"
    movel(Linea21_AB_p, a=0.5, v=0.1)
    $ 4222 "bajada_comprobacion"
    $ 4223 "Direction: Base Z-"
    global move_thread_flag_4223=0
    thread move_thread_4223():
      enter_critical
      move_thread_flag_4223 = 1
      local towardsPos=calculate_point_to_move_towards(p[0.0,0.0,0.0,0.0,0.0,0.0], [0.0,0.0,-1.0], 0.071)
      movel(towardsPos, a=0.15, v=0.1)
      move_thread_flag_4223 = 2
      exit_critical
    end
    move_thread_flag_4223 = 0
    move_thread_han_4223 = run move_thread_4223()
    while (True):
      sleep(1.0E-10)
      if (move_thread_flag_4223 > 1):
        join move_thread_han_4223
        $ 4224 "Until (distance)"
        break
      end
      sync()
    end
    $ 4225 "Direction: Base Z-"
    global move_thread_flag_4225=0
    thread move_thread_4225():
      enter_critical
      move_thread_flag_4225 = 1
      local towardsPos=calculate_point_to_move_towards(p[0.0,0.0,0.0,0.0,0.0,0.0], [0.0,0.0,-1.0], 1000.0)
      movel(towardsPos, a=0.007, v=0.007)
      move_thread_flag_4225 = 2
      exit_critical
    end
    move_thread_flag_4225 = 0
    move_thread_han_4225 = run move_thread_4225()
    while (True):
      local targetTcpDirection=get_target_tcp_speed()
      local stepsToRetract=tool_contact(direction=targetTcpDirection)
      if (stepsToRetract > 0):
        kill move_thread_han_4225
        stopl(0.02)
        local backTrackMovement=get_actual_joint_positions_history(stepsToRetract)
        local contactPose=get_forward_kin(backTrackMovement)
        local posDir=[targetTcpDirection[0],targetTcpDirection[1],targetTcpDirection[2]]
        local retractTo=contactPose
        if (norm(posDir) > 1e-6):
          local normalizedPosDir=normalize(posDir)
          local additionalRetraction=p[normalizedPosDir[0] * 0.0, normalizedPosDir[1] * 0.0, normalizedPosDir[2] * 0.0, 0, 0, 0]
          retractTo = pose_sub(contactPose, additionalRetraction)
        end
        movel(retractTo, a=0.02, v=0.1)
        $ 4226 "Until (tool_contact_detection)"
        break
      end
      sync()
    end
    $ 4227 "Direction: Base Z+"
    global move_thread_flag_4227=0
    thread move_thread_4227():
      enter_critical
      move_thread_flag_4227 = 1
      local towardsPos=calculate_point_to_move_towards(p[0.0,0.0,0.0,0.0,0.0,0.0], [0.0,0.0,1.0], 0.08)
      movel(towardsPos, a=0.15, v=0.1)
      move_thread_flag_4227 = 2
      exit_critical
    end
    move_thread_flag_4227 = 0
    move_thread_han_4227 = run move_thread_4227()
    while (True):
      sleep(1.0E-10)
      if (move_thread_flag_4227 > 1):
        join move_thread_han_4227
        $ 4228 "Until (distance)"
        break
      end
      sync()
    end
    $ 4229 "AB"
    $ 4230 "'desbaste_inicial'"
    # 'desbaste_inicial'
    $ 4231 "bajada_broca≔p[0,0,-0.008,0,0,0]"
    global bajada_broca=p[0,0,-0.008,0,0,0]
    $ 4232 "barrenos_menos1≔12"
    global barrenos_menos1=12
    $ 4233 "barreno_actual≔0"
    global barreno_actual=0
    $ 4234 "Loop barreno_actual≤barrenos_menos1"
    while (barreno_actual <= barrenos_menos1):
      $ 4235 "Perforacion"
      $ 4236 "MoveL"
      $ 4237 "If barreno_actual≟6"
      if (barreno_actual == 6):
        $ 4238 "barreno_actual≔barreno_actual+1"
        global barreno_actual=barreno_actual+1
      end
      $ 4239 "internos≔interpolate_pose(Linea21_A, Linea21_AB, barreno_actual/barrenos_menos1)"
      global internos= interpolate_pose (Linea21_A_p, Linea21_AB_p, barreno_actual/barrenos_menos1)
      $ 4240 "internos" "breakAfter"
      movel(internos, a=0.5, v=0.1)
      $ 4241 "'desbaste_inicial'"
      # 'desbaste_inicial'
      $ 4242 "bajada_broca≔p[0,0,-0.024,0,0,0]"
      global bajada_broca=p[0,0,-0.024,0,0,0]
      $ 4243 "bajada≔p[0,0,0.024,0,0,0]"
      global bajada=p[0,0,0.024,0,0,0]
      $ 4244 "Direction: Base Z-"
      global move_thread_flag_4244=0
      thread move_thread_4244():
        enter_critical
        move_thread_flag_4244 = 1
        local towardsPos=calculate_point_to_move_towards(p[0.0,0.0,0.0,0.0,0.0,0.0], [0.0,0.0,-1.0], 0.071)
        movel(towardsPos, a=0.15, v=0.1)
        move_thread_flag_4244 = 2
        exit_critical
      end
      move_thread_flag_4244 = 0
      move_thread_han_4244 = run move_thread_4244()
      while (True):
        sleep(1.0E-10)
        if (move_thread_flag_4244 > 1):
          join move_thread_han_4244
          $ 4245 "Until (distance)"
          break
        end
        sync()
      end
      $ 4246 "Direction: Base Z-"
      global move_thread_flag_4246=0
      thread move_thread_4246():
        enter_critical
        move_thread_flag_4246 = 1
        local towardsPos=calculate_point_to_move_towards(p[0.0,0.0,0.0,0.0,0.0,0.0], [0.0,0.0,-1.0], 1000.0)
        movel(towardsPos, a=0.007, v=0.007)
        move_thread_flag_4246 = 2
        exit_critical
      end
      move_thread_flag_4246 = 0
      move_thread_han_4246 = run move_thread_4246()
      while (True):
        local targetTcpDirection=get_target_tcp_speed()
        local stepsToRetract=tool_contact(direction=targetTcpDirection)
        if (stepsToRetract > 0):
          kill move_thread_han_4246
          stopl(0.02)
          local backTrackMovement=get_actual_joint_positions_history(stepsToRetract)
          local contactPose=get_forward_kin(backTrackMovement)
          local posDir=[targetTcpDirection[0],targetTcpDirection[1],targetTcpDirection[2]]
          local retractTo=contactPose
          if (norm(posDir) > 1e-6):
            local normalizedPosDir=normalize(posDir)
            local additionalRetraction=p[normalizedPosDir[0] * 0.0, normalizedPosDir[1] * 0.0, normalizedPosDir[2] * 0.0, 0, 0, 0]
            retractTo = pose_sub(contactPose, additionalRetraction)
          end
          movel(retractTo, a=0.02, v=0.1)
          $ 4247 "Until (tool_contact_detection)"
          break
        end
        sync()
      end
      $ 4248 "Popup: punto contacto alanzdo"
      popup("punto contacto alanzdo", "Mensaje", False, False, blocking=True)
      $ 4249 "Direction: Base Z+"
      global move_thread_flag_4249=0
      thread move_thread_4249():
        enter_critical
        move_thread_flag_4249 = 1
        local towardsPos=calculate_point_to_move_towards(p[0.0,0.0,0.0,0.0,0.0,0.0], [0.0,0.0,1.0], 0.007)
        movel(towardsPos, a=0.015, v=0.015)
        move_thread_flag_4249 = 2
        exit_critical
      end
      move_thread_flag_4249 = 0
      move_thread_han_4249 = run move_thread_4249()
      while (True):
        sleep(1.0E-10)
        if (move_thread_flag_4249 > 1):
          join move_thread_han_4249
          $ 4250 "Until (distance)"
          break
        end
        sync()
      end
      $ 4251 "Wait: 0.3"
      sleep(0.3)
      $ 4252 "Set CO[1]=Encender"
      set_configurable_digital_out(1, True)
      $ 4253 "Wait: 0.3"
      sleep(0.3)
      $ 4254 "Loop 1 times"
      Loop_76 = 0
      while (Loop_76 < 1):
        $ 4255 "bajar≔pose_add(get_actual_tcp_pose(), bajada_broca)"
        global bajar= pose_add ( get_actual_tcp_pose (), bajada_broca)
        $ 4256 "bajar" "breakAfter"
        movel(bajar, a=0.004, v=0.004)
        $ 4257 "subir≔pose_sub(get_actual_tcp_pose(), bajada_broca)"
        global subir= pose_sub ( get_actual_tcp_pose (), bajada_broca)
        $ 4258 "Direction: Base Z+"
        global move_thread_flag_4258=0
        thread move_thread_4258():
          enter_critical
          move_thread_flag_4258 = 1
          local towardsPos=calculate_point_to_move_towards(p[0.0,0.0,0.0,0.0,0.0,0.0], [0.0,0.0,1.0], 0.002)
          movel(towardsPos, a=0.015, v=0.015)
          move_thread_flag_4258 = 2
          exit_critical
        end
        move_thread_flag_4258 = 0
        move_thread_han_4258 = run move_thread_4258()
        while (True):
          sleep(1.0E-10)
          if (move_thread_flag_4258 > 1):
            join move_thread_han_4258
            $ 4259 "Until (distance)"
            break
          end
          sync()
        end
        $ 4260 "Set CO[1]=Apagar"
        set_configurable_digital_out(1, False)
        $ 4261 "subir" "breakAfter"
        movel(subir, a=0.015, v=0.015)
        $ 4262 "bajada_broca≔pose_sub(bajada_broca, bajada)"
        global bajada_broca= pose_sub (bajada_broca, bajada)
        Loop_76 = Loop_76 + 1
      end
      $ 4263 "Direction: Base Z+"
      global move_thread_flag_4263=0
      thread move_thread_4263():
        enter_critical
        move_thread_flag_4263 = 1
        local towardsPos=calculate_point_to_move_towards(p[0.0,0.0,0.0,0.0,0.0,0.0], [0.0,0.0,1.0], 0.08)
        movel(towardsPos, a=0.15, v=0.1)
        move_thread_flag_4263 = 2
        exit_critical
      end
      move_thread_flag_4263 = 0
      move_thread_han_4263 = run move_thread_4263()
      while (True):
        sleep(1.0E-10)
        if (move_thread_flag_4263 > 1):
          join move_thread_han_4263
          $ 4264 "Until (distance)"
          break
        end
        sync()
      end
      $ 4265 "Set CO[1]=Apagar"
      set_configurable_digital_out(1, False)
      $ 4266 "barreno_actual≔barreno_actual+1"
      global barreno_actual=barreno_actual+1
    end
    $ 4269 "Popup: Linea21 con chica Terminada!"
    popup("Linea21 con chica Terminada!", "Mensaje", False, False, blocking=True)
    $ 4270 "Linea21B"
    $ 4271 "Marcar_puntos"
    $ 4272 "MoveL"
    $ 4274 "Linea21_BA" "breakAfter"
    movel(Linea21_BA_p, a=0.5, v=0.1)
    $ 4275 "bajada_comprobacion"
    $ 4276 "Direction: Base Z-"
    global move_thread_flag_4276=0
    thread move_thread_4276():
      enter_critical
      move_thread_flag_4276 = 1
      local towardsPos=calculate_point_to_move_towards(p[0.0,0.0,0.0,0.0,0.0,0.0], [0.0,0.0,-1.0], 0.071)
      movel(towardsPos, a=0.15, v=0.1)
      move_thread_flag_4276 = 2
      exit_critical
    end
    move_thread_flag_4276 = 0
    move_thread_han_4276 = run move_thread_4276()
    while (True):
      sleep(1.0E-10)
      if (move_thread_flag_4276 > 1):
        join move_thread_han_4276
        $ 4277 "Until (distance)"
        break
      end
      sync()
    end
    $ 4278 "Direction: Base Z-"
    global move_thread_flag_4278=0
    thread move_thread_4278():
      enter_critical
      move_thread_flag_4278 = 1
      local towardsPos=calculate_point_to_move_towards(p[0.0,0.0,0.0,0.0,0.0,0.0], [0.0,0.0,-1.0], 1000.0)
      movel(towardsPos, a=0.007, v=0.007)
      move_thread_flag_4278 = 2
      exit_critical
    end
    move_thread_flag_4278 = 0
    move_thread_han_4278 = run move_thread_4278()
    while (True):
      local targetTcpDirection=get_target_tcp_speed()
      local stepsToRetract=tool_contact(direction=targetTcpDirection)
      if (stepsToRetract > 0):
        kill move_thread_han_4278
        stopl(0.02)
        local backTrackMovement=get_actual_joint_positions_history(stepsToRetract)
        local contactPose=get_forward_kin(backTrackMovement)
        local posDir=[targetTcpDirection[0],targetTcpDirection[1],targetTcpDirection[2]]
        local retractTo=contactPose
        if (norm(posDir) > 1e-6):
          local normalizedPosDir=normalize(posDir)
          local additionalRetraction=p[normalizedPosDir[0] * 0.0, normalizedPosDir[1] * 0.0, normalizedPosDir[2] * 0.0, 0, 0, 0]
          retractTo = pose_sub(contactPose, additionalRetraction)
        end
        movel(retractTo, a=0.02, v=0.1)
        $ 4279 "Until (tool_contact_detection)"
        break
      end
      sync()
    end
    $ 4280 "Direction: Base Z+"
    global move_thread_flag_4280=0
    thread move_thread_4280():
      enter_critical
      move_thread_flag_4280 = 1
      local towardsPos=calculate_point_to_move_towards(p[0.0,0.0,0.0,0.0,0.0,0.0], [0.0,0.0,1.0], 0.08)
      movel(towardsPos, a=0.15, v=0.1)
      move_thread_flag_4280 = 2
      exit_critical
    end
    move_thread_flag_4280 = 0
    move_thread_han_4280 = run move_thread_4280()
    while (True):
      sleep(1.0E-10)
      if (move_thread_flag_4280 > 1):
        join move_thread_han_4280
        $ 4281 "Until (distance)"
        break
      end
      sync()
    end
    $ 4283 "Linea21_B" "breakAfter"
    movel(Linea21_B_p, a=0.5, v=0.1)
    $ 4284 "bajada_comprobacion"
    $ 4285 "Direction: Base Z-"
    global move_thread_flag_4285=0
    thread move_thread_4285():
      enter_critical
      move_thread_flag_4285 = 1
      local towardsPos=calculate_point_to_move_towards(p[0.0,0.0,0.0,0.0,0.0,0.0], [0.0,0.0,-1.0], 0.071)
      movel(towardsPos, a=0.15, v=0.1)
      move_thread_flag_4285 = 2
      exit_critical
    end
    move_thread_flag_4285 = 0
    move_thread_han_4285 = run move_thread_4285()
    while (True):
      sleep(1.0E-10)
      if (move_thread_flag_4285 > 1):
        join move_thread_han_4285
        $ 4286 "Until (distance)"
        break
      end
      sync()
    end
    $ 4287 "Direction: Base Z-"
    global move_thread_flag_4287=0
    thread move_thread_4287():
      enter_critical
      move_thread_flag_4287 = 1
      local towardsPos=calculate_point_to_move_towards(p[0.0,0.0,0.0,0.0,0.0,0.0], [0.0,0.0,-1.0], 1000.0)
      movel(towardsPos, a=0.007, v=0.007)
      move_thread_flag_4287 = 2
      exit_critical
    end
    move_thread_flag_4287 = 0
    move_thread_han_4287 = run move_thread_4287()
    while (True):
      local targetTcpDirection=get_target_tcp_speed()
      local stepsToRetract=tool_contact(direction=targetTcpDirection)
      if (stepsToRetract > 0):
        kill move_thread_han_4287
        stopl(0.02)
        local backTrackMovement=get_actual_joint_positions_history(stepsToRetract)
        local contactPose=get_forward_kin(backTrackMovement)
        local posDir=[targetTcpDirection[0],targetTcpDirection[1],targetTcpDirection[2]]
        local retractTo=contactPose
        if (norm(posDir) > 1e-6):
          local normalizedPosDir=normalize(posDir)
          local additionalRetraction=p[normalizedPosDir[0] * 0.0, normalizedPosDir[1] * 0.0, normalizedPosDir[2] * 0.0, 0, 0, 0]
          retractTo = pose_sub(contactPose, additionalRetraction)
        end
        movel(retractTo, a=0.02, v=0.1)
        $ 4288 "Until (tool_contact_detection)"
        break
      end
      sync()
    end
    $ 4289 "Direction: Base Z+"
    global move_thread_flag_4289=0
    thread move_thread_4289():
      enter_critical
      move_thread_flag_4289 = 1
      local towardsPos=calculate_point_to_move_towards(p[0.0,0.0,0.0,0.0,0.0,0.0], [0.0,0.0,1.0], 0.08)
      movel(towardsPos, a=0.15, v=0.1)
      move_thread_flag_4289 = 2
      exit_critical
    end
    move_thread_flag_4289 = 0
    move_thread_han_4289 = run move_thread_4289()
    while (True):
      sleep(1.0E-10)
      if (move_thread_flag_4289 > 1):
        join move_thread_han_4289
        $ 4290 "Until (distance)"
        break
      end
      sync()
    end
    $ 4291 "AB"
    $ 4292 "'desbaste_inicial'"
    # 'desbaste_inicial'
    $ 4293 "bajada_broca≔p[0,0,-0.008,0,0,0]"
    global bajada_broca=p[0,0,-0.008,0,0,0]
    $ 4294 "barrenos_menos1≔5"
    global barrenos_menos1=5
    $ 4295 "barreno_actual≔0"
    global barreno_actual=0
    $ 4296 "Loop barreno_actual≤barrenos_menos1"
    while (barreno_actual <= barrenos_menos1):
      $ 4297 "Perforacion"
      $ 4298 "MoveL"
      $ 4301 "internos≔interpolate_pose(Linea21_BA, Linea21_B, barreno_actual/barrenos_menos1)"
      global internos= interpolate_pose (Linea21_BA_p, Linea21_B_p, barreno_actual/barrenos_menos1)
      $ 4302 "internos" "breakAfter"
      movel(internos, a=0.5, v=0.1)
      $ 4303 "'desbaste_inicial'"
      # 'desbaste_inicial'
      $ 4304 "bajada_broca≔p[0,0,-0.024,0,0,0]"
      global bajada_broca=p[0,0,-0.024,0,0,0]
      $ 4305 "bajada≔p[0,0,0.024,0,0,0]"
      global bajada=p[0,0,0.024,0,0,0]
      $ 4306 "Direction: Base Z-"
      global move_thread_flag_4306=0
      thread move_thread_4306():
        enter_critical
        move_thread_flag_4306 = 1
        local towardsPos=calculate_point_to_move_towards(p[0.0,0.0,0.0,0.0,0.0,0.0], [0.0,0.0,-1.0], 0.071)
        movel(towardsPos, a=0.15, v=0.1)
        move_thread_flag_4306 = 2
        exit_critical
      end
